REGION Network 6
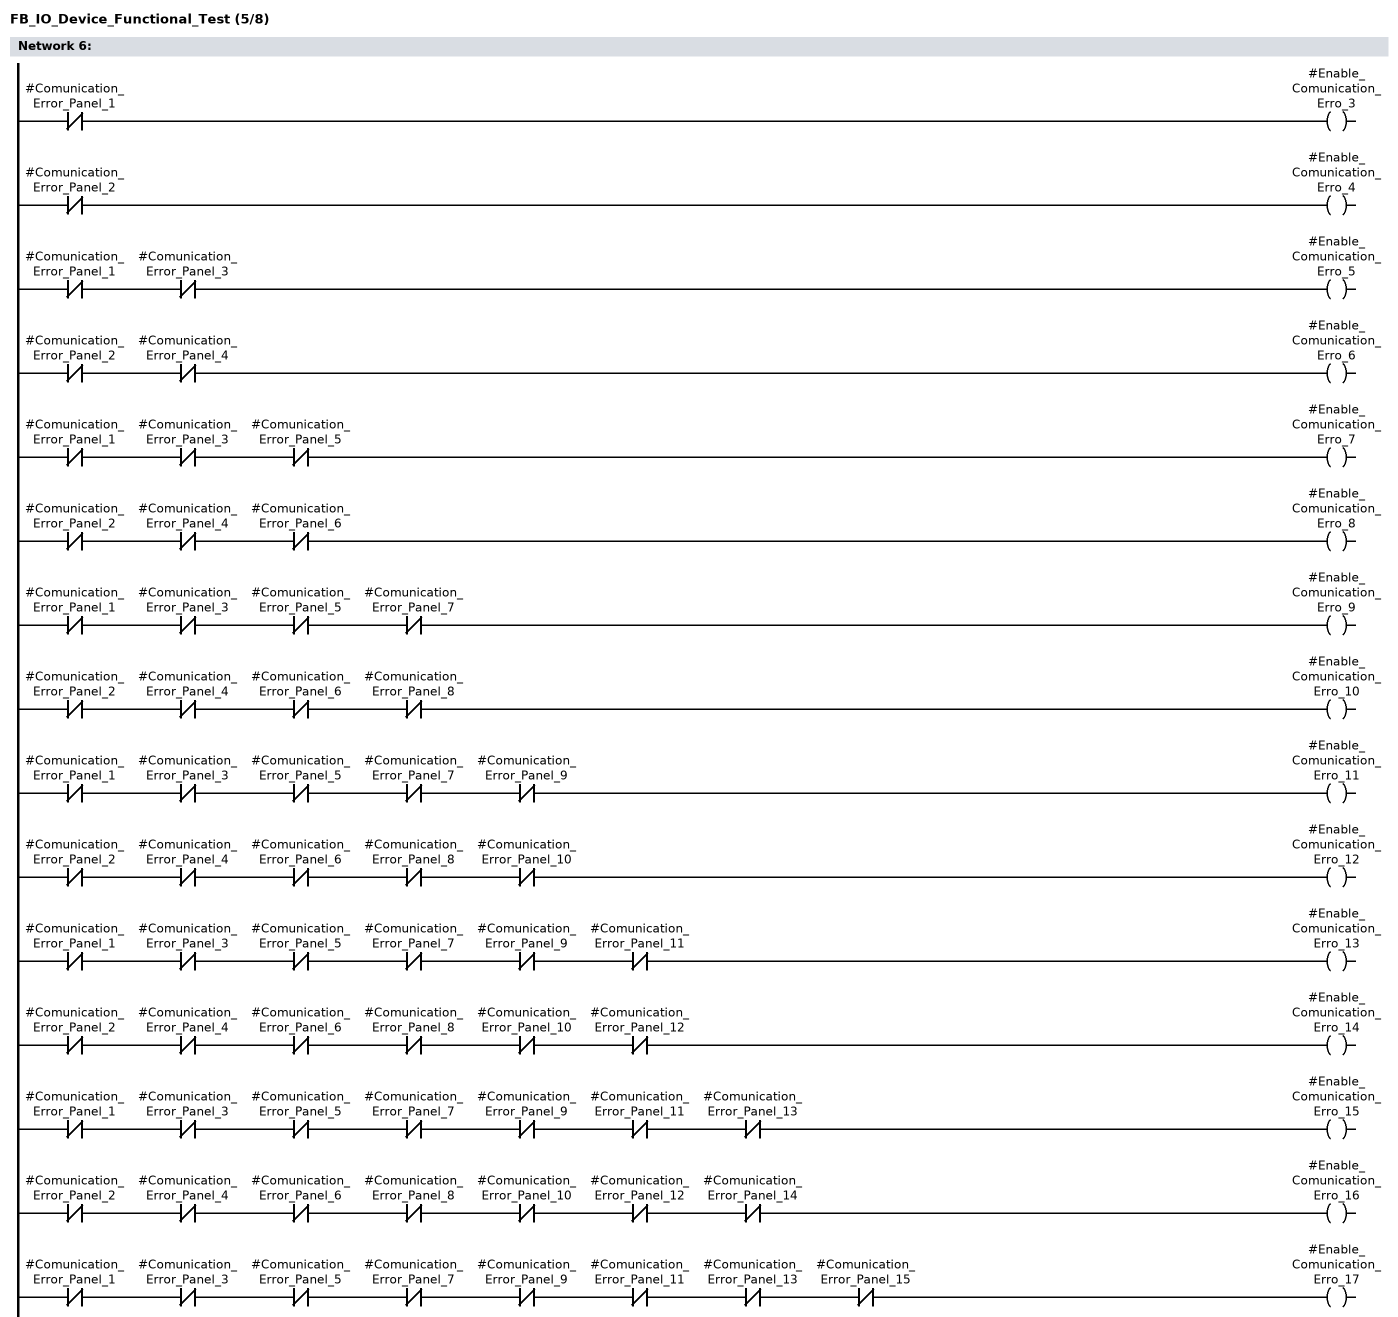
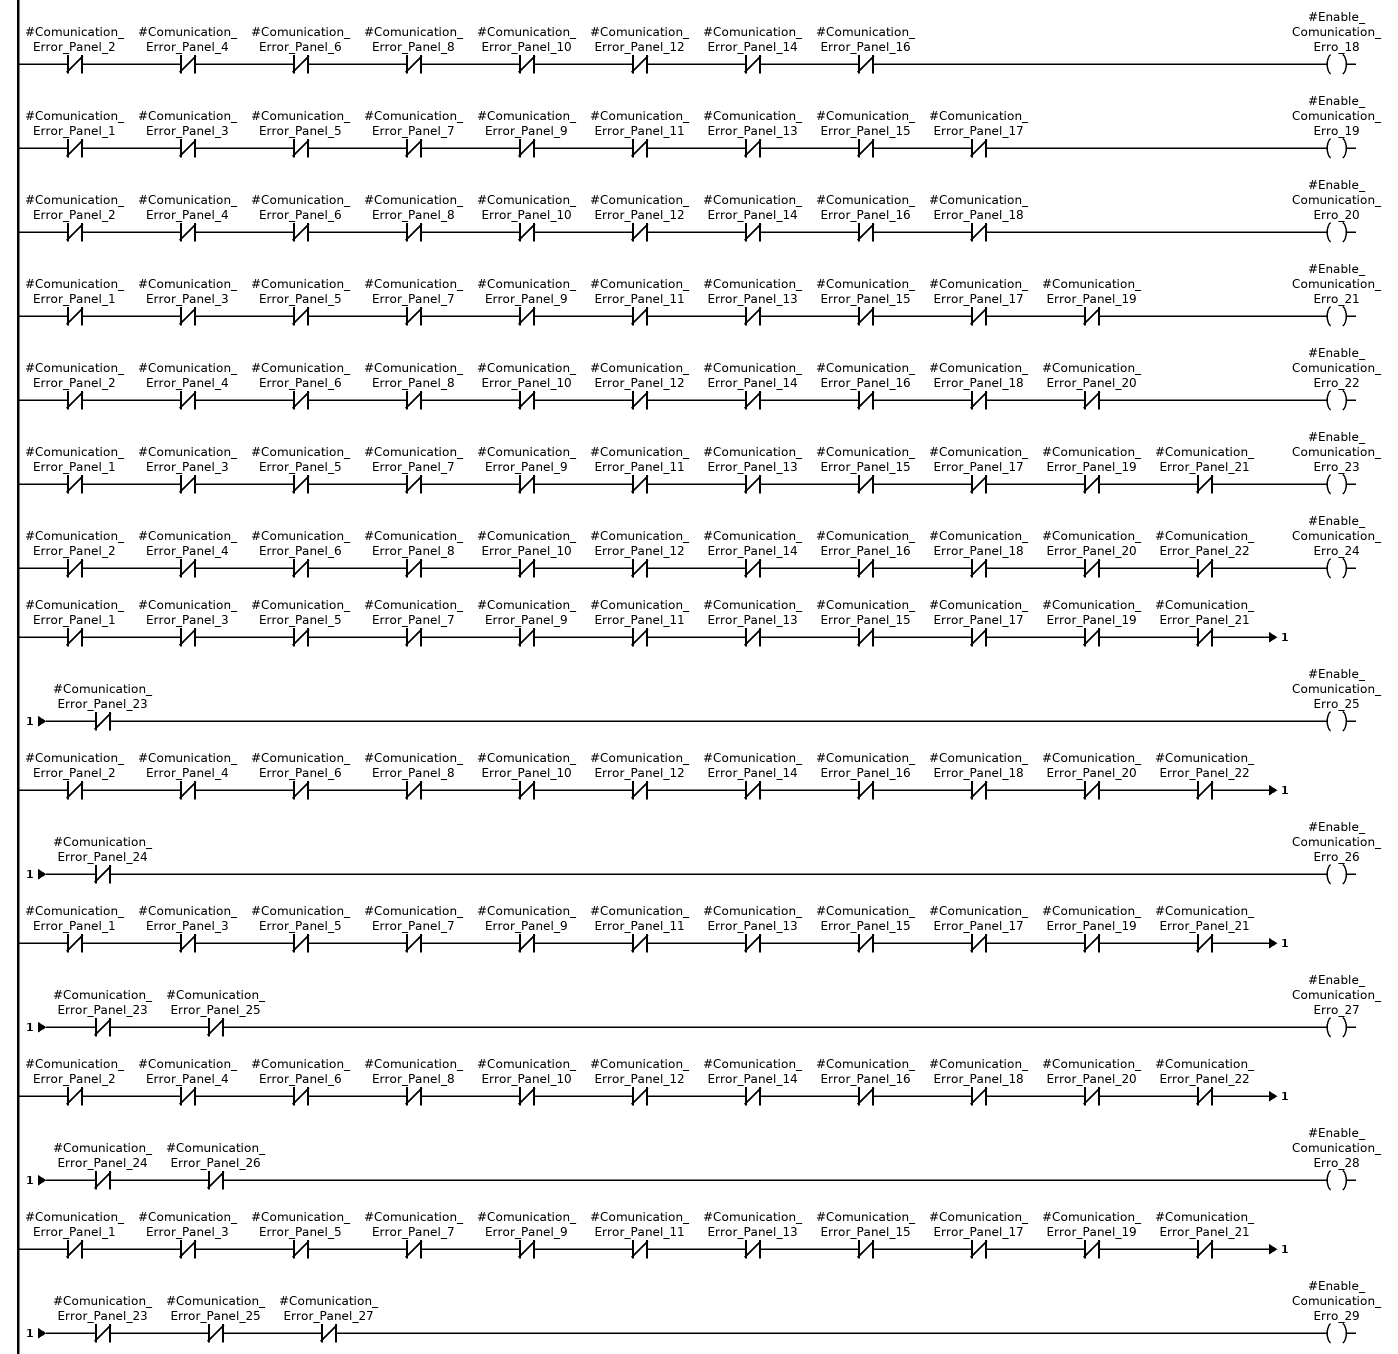
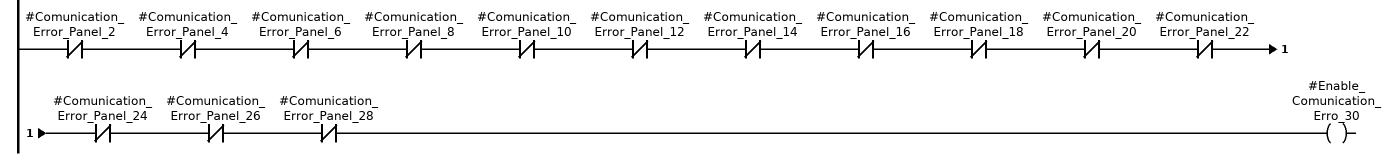
   RUNG wire#powerrail
      I_Contact( #Comunication_Error_Panel_1 )
      Coil( #Enable_Comunication_Erro_3 )
   END_RUNG
   RUNG wire#powerrail
      I_Contact( #Comunication_Error_Panel_2 )
      Coil( #Enable_Comunication_Erro_4 )
   END_RUNG
   RUNG wire#powerrail
      I_Contact( #Comunication_Error_Panel_1 )
      I_Contact( #Comunication_Error_Panel_3 )
      Coil( #Enable_Comunication_Erro_5 )
   END_RUNG
   RUNG wire#powerrail
      I_Contact( #Comunication_Error_Panel_2 )
      I_Contact( #Comunication_Error_Panel_4 )
      Coil( #Enable_Comunication_Erro_6 )
   END_RUNG
   RUNG wire#powerrail
      I_Contact( #Comunication_Error_Panel_1 )
      I_Contact( #Comunication_Error_Panel_3 )
      I_Contact( #Comunication_Error_Panel_5 )
      Coil( #Enable_Comunication_Erro_7 )
   END_RUNG
   RUNG wire#powerrail
      I_Contact( #Comunication_Error_Panel_2 )
      I_Contact( #Comunication_Error_Panel_4 )
      I_Contact( #Comunication_Error_Panel_6 )
      Coil( #Enable_Comunication_Erro_8 )
   END_RUNG
   RUNG wire#powerrail
      I_Contact( #Comunication_Error_Panel_1 )
      I_Contact( #Comunication_Error_Panel_3 )
      I_Contact( #Comunication_Error_Panel_5 )
      I_Contact( #Comunication_Error_Panel_7 )
      Coil( #Enable_Comunication_Erro_9 )
   END_RUNG
   RUNG wire#powerrail
      I_Contact( #Comunication_Error_Panel_2 )
      I_Contact( #Comunication_Error_Panel_4 )
      I_Contact( #Comunication_Error_Panel_6 )
      I_Contact( #Comunication_Error_Panel_8 )
      Coil( #Enable_Comunication_Erro_10 )
   END_RUNG
   RUNG wire#powerrail
      I_Contact( #Comunication_Error_Panel_1 )
      I_Contact( #Comunication_Error_Panel_3 )
      I_Contact( #Comunication_Error_Panel_5 )
      I_Contact( #Comunication_Error_Panel_7 )
      I_Contact( #Comunication_Error_Panel_9 )
      Coil( #Enable_Comunication_Erro_11 )
   END_RUNG
   RUNG wire#powerrail
      I_Contact( #Comunication_Error_Panel_2 )
      I_Contact( #Comunication_Error_Panel_4 )
      I_Contact( #Comunication_Error_Panel_6 )
      I_Contact( #Comunication_Error_Panel_8 )
      I_Contact( #Comunication_Error_Panel_10 )
      Coil( #Enable_Comunication_Erro_12 )
   END_RUNG
   RUNG wire#powerrail
      I_Contact( #Comunication_Error_Panel_1 )
      I_Contact( #Comunication_Error_Panel_3 )
      I_Contact( #Comunication_Error_Panel_5 )
      I_Contact( #Comunication_Error_Panel_7 )
      I_Contact( #Comunication_Error_Panel_9 )
      I_Contact( #Comunication_Error_Panel_11 )
      Coil( #Enable_Comunication_Erro_13 )
   END_RUNG
   RUNG wire#powerrail
      I_Contact( #Comunication_Error_Panel_2 )
      I_Contact( #Comunication_Error_Panel_4 )
      I_Contact( #Comunication_Error_Panel_6 )
      I_Contact( #Comunication_Error_Panel_8 )
      I_Contact( #Comunication_Error_Panel_10 )
      I_Contact( #Comunication_Error_Panel_12 )
      Coil( #Enable_Comunication_Erro_14 )
   END_RUNG
   RUNG wire#powerrail
      I_Contact( #Comunication_Error_Panel_1 )
      I_Contact( #Comunication_Error_Panel_3 )
      I_Contact( #Comunication_Error_Panel_5 )
      I_Contact( #Comunication_Error_Panel_7 )
      I_Contact( #Comunication_Error_Panel_9 )
      I_Contact( #Comunication_Error_Panel_11 )
      I_Contact( #Comunication_Error_Panel_13 )
      Coil( #Enable_Comunication_Erro_15 )
   END_RUNG
   RUNG wire#powerrail
      I_Contact( #Comunication_Error_Panel_2 )
      I_Contact( #Comunication_Error_Panel_4 )
      I_Contact( #Comunication_Error_Panel_6 )
      I_Contact( #Comunication_Error_Panel_8 )
      I_Contact( #Comunication_Error_Panel_10 )
      I_Contact( #Comunication_Error_Panel_12 )
      I_Contact( #Comunication_Error_Panel_14 )
      Coil( #Enable_Comunication_Erro_16 )
   END_RUNG
   RUNG wire#powerrail
      I_Contact( #Comunication_Error_Panel_1 )
      I_Contact( #Comunication_Error_Panel_3 )
      I_Contact( #Comunication_Error_Panel_5 )
      I_Contact( #Comunication_Error_Panel_7 )
      I_Contact( #Comunication_Error_Panel_9 )
      I_Contact( #Comunication_Error_Panel_11 )
      I_Contact( #Comunication_Error_Panel_13 )
      I_Contact( #Comunication_Error_Panel_15 )
      Coil( #Enable_Comunication_Erro_17 )
   END_RUNG
   RUNG wire#powerrail
      I_Contact( #Comunication_Error_Panel_2 )
      I_Contact( #Comunication_Error_Panel_4 )
      I_Contact( #Comunication_Error_Panel_6 )
      I_Contact( #Comunication_Error_Panel_8 )
      I_Contact( #Comunication_Error_Panel_10 )
      I_Contact( #Comunication_Error_Panel_12 )
      I_Contact( #Comunication_Error_Panel_14 )
      I_Contact( #Comunication_Error_Panel_16 )
      Coil( #Enable_Comunication_Erro_18 )
   END_RUNG
   RUNG wire#powerrail
      I_Contact( #Comunication_Error_Panel_1 )
      I_Contact( #Comunication_Error_Panel_3 )
      I_Contact( #Comunication_Error_Panel_5 )
      I_Contact( #Comunication_Error_Panel_7 )
      I_Contact( #Comunication_Error_Panel_9 )
      I_Contact( #Comunication_Error_Panel_11 )
      I_Contact( #Comunication_Error_Panel_13 )
      I_Contact( #Comunication_Error_Panel_15 )
      I_Contact( #Comunication_Error_Panel_17 )
      Coil( #Enable_Comunication_Erro_19 )
   END_RUNG
   RUNG wire#powerrail
      I_Contact( #Comunication_Error_Panel_2 )
      I_Contact( #Comunication_Error_Panel_4 )
      I_Contact( #Comunication_Error_Panel_6 )
      I_Contact( #Comunication_Error_Panel_8 )
      I_Contact( #Comunication_Error_Panel_10 )
      I_Contact( #Comunication_Error_Panel_12 )
      I_Contact( #Comunication_Error_Panel_14 )
      I_Contact( #Comunication_Error_Panel_16 )
      I_Contact( #Comunication_Error_Panel_18 )
      Coil( #Enable_Comunication_Erro_20 )
   END_RUNG
   RUNG wire#powerrail
      I_Contact( #Comunication_Error_Panel_1 )
      I_Contact( #Comunication_Error_Panel_3 )
      I_Contact( #Comunication_Error_Panel_5 )
      I_Contact( #Comunication_Error_Panel_7 )
      I_Contact( #Comunication_Error_Panel_9 )
      I_Contact( #Comunication_Error_Panel_11 )
      I_Contact( #Comunication_Error_Panel_13 )
      I_Contact( #Comunication_Error_Panel_15 )
      I_Contact( #Comunication_Error_Panel_17 )
      I_Contact( #Comunication_Error_Panel_19 )
      Coil( #Enable_Comunication_Erro_21 )
   END_RUNG
   RUNG wire#powerrail
      I_Contact( #Comunication_Error_Panel_2 )
      I_Contact( #Comunication_Error_Panel_4 )
      I_Contact( #Comunication_Error_Panel_6 )
      I_Contact( #Comunication_Error_Panel_8 )
      I_Contact( #Comunication_Error_Panel_10 )
      I_Contact( #Comunication_Error_Panel_12 )
      I_Contact( #Comunication_Error_Panel_14 )
      I_Contact( #Comunication_Error_Panel_16 )
      I_Contact( #Comunication_Error_Panel_18 )
      I_Contact( #Comunication_Error_Panel_20 )
      Coil( #Enable_Comunication_Erro_22 )
   END_RUNG
   RUNG wire#powerrail
      I_Contact( #Comunication_Error_Panel_1 )
      I_Contact( #Comunication_Error_Panel_3 )
      I_Contact( #Comunication_Error_Panel_5 )
      I_Contact( #Comunication_Error_Panel_7 )
      I_Contact( #Comunication_Error_Panel_9 )
      I_Contact( #Comunication_Error_Panel_11 )
      I_Contact( #Comunication_Error_Panel_13 )
      I_Contact( #Comunication_Error_Panel_15 )
      I_Contact( #Comunication_Error_Panel_17 )
      I_Contact( #Comunication_Error_Panel_19 )
      I_Contact( #Comunication_Error_Panel_21 )
      Coil( #Enable_Comunication_Erro_23 )
   END_RUNG
   RUNG wire#powerrail
      I_Contact( #Comunication_Error_Panel_2 )
      I_Contact( #Comunication_Error_Panel_4 )
      I_Contact( #Comunication_Error_Panel_6 )
      I_Contact( #Comunication_Error_Panel_8 )
      I_Contact( #Comunication_Error_Panel_10 )
      I_Contact( #Comunication_Error_Panel_12 )
      I_Contact( #Comunication_Error_Panel_14 )
      I_Contact( #Comunication_Error_Panel_16 )
      I_Contact( #Comunication_Error_Panel_18 )
      I_Contact( #Comunication_Error_Panel_20 )
      I_Contact( #Comunication_Error_Panel_22 )
      Coil( #Enable_Comunication_Erro_24 )
   END_RUNG
   RUNG wire#powerrail
      I_Contact( #Comunication_Error_Panel_1 )
      I_Contact( #Comunication_Error_Panel_3 )
      I_Contact( #Comunication_Error_Panel_5 )
      I_Contact( #Comunication_Error_Panel_7 )
      I_Contact( #Comunication_Error_Panel_9 )
      I_Contact( #Comunication_Error_Panel_11 )
      I_Contact( #Comunication_Error_Panel_13 )
      I_Contact( #Comunication_Error_Panel_15 )
      I_Contact( #Comunication_Error_Panel_17 )
      I_Contact( #Comunication_Error_Panel_19 )
      I_Contact( #Comunication_Error_Panel_21 )
      I_Contact( #Comunication_Error_Panel_23 )
      Coil( #Enable_Comunication_Erro_25 )
   END_RUNG
   RUNG wire#powerrail
      I_Contact( #Comunication_Error_Panel_2 )
      I_Contact( #Comunication_Error_Panel_4 )
      I_Contact( #Comunication_Error_Panel_6 )
      I_Contact( #Comunication_Error_Panel_8 )
      I_Contact( #Comunication_Error_Panel_10 )
      I_Contact( #Comunication_Error_Panel_12 )
      I_Contact( #Comunication_Error_Panel_14 )
      I_Contact( #Comunication_Error_Panel_16 )
      I_Contact( #Comunication_Error_Panel_18 )
      I_Contact( #Comunication_Error_Panel_20 )
      I_Contact( #Comunication_Error_Panel_22 )
      I_Contact( #Comunication_Error_Panel_24 )
      Coil( #Enable_Comunication_Erro_26 )
   END_RUNG
   RUNG wire#powerrail
      I_Contact( #Comunication_Error_Panel_1 )
      I_Contact( #Comunication_Error_Panel_3 )
      I_Contact( #Comunication_Error_Panel_5 )
      I_Contact( #Comunication_Error_Panel_7 )
      I_Contact( #Comunication_Error_Panel_9 )
      I_Contact( #Comunication_Error_Panel_11 )
      I_Contact( #Comunication_Error_Panel_13 )
      I_Contact( #Comunication_Error_Panel_15 )
      I_Contact( #Comunication_Error_Panel_17 )
      I_Contact( #Comunication_Error_Panel_19 )
      I_Contact( #Comunication_Error_Panel_21 )
      I_Contact( #Comunication_Error_Panel_23 )
      I_Contact( #Comunication_Error_Panel_25 )
      Coil( #Enable_Comunication_Erro_27 )
   END_RUNG
   RUNG wire#powerrail
      I_Contact( #Comunication_Error_Panel_2 )
      I_Contact( #Comunication_Error_Panel_4 )
      I_Contact( #Comunication_Error_Panel_6 )
      I_Contact( #Comunication_Error_Panel_8 )
      I_Contact( #Comunication_Error_Panel_10 )
      I_Contact( #Comunication_Error_Panel_12 )
      I_Contact( #Comunication_Error_Panel_14 )
      I_Contact( #Comunication_Error_Panel_16 )
      I_Contact( #Comunication_Error_Panel_18 )
      I_Contact( #Comunication_Error_Panel_20 )
      I_Contact( #Comunication_Error_Panel_22 )
      I_Contact( #Comunication_Error_Panel_24 )
      I_Contact( #Comunication_Error_Panel_26 )
      Coil( #Enable_Comunication_Erro_28 )
   END_RUNG
   RUNG wire#powerrail
      I_Contact( #Comunication_Error_Panel_1 )
      I_Contact( #Comunication_Error_Panel_3 )
      I_Contact( #Comunication_Error_Panel_5 )
      I_Contact( #Comunication_Error_Panel_7 )
      I_Contact( #Comunication_Error_Panel_9 )
      I_Contact( #Comunication_Error_Panel_11 )
      I_Contact( #Comunication_Error_Panel_13 )
      I_Contact( #Comunication_Error_Panel_15 )
      I_Contact( #Comunication_Error_Panel_17 )
      I_Contact( #Comunication_Error_Panel_19 )
      I_Contact( #Comunication_Error_Panel_21 )
      I_Contact( #Comunication_Error_Panel_23 )
      I_Contact( #Comunication_Error_Panel_25 )
      I_Contact( #Comunication_Error_Panel_27 )
      Coil( #Enable_Comunication_Erro_29 )
   END_RUNG
   RUNG wire#powerrail
      I_Contact( #Comunication_Error_Panel_2 )
      I_Contact( #Comunication_Error_Panel_4 )
      I_Contact( #Comunication_Error_Panel_6 )
      I_Contact( #Comunication_Error_Panel_8 )
      I_Contact( #Comunication_Error_Panel_10 )
      I_Contact( #Comunication_Error_Panel_12 )
      I_Contact( #Comunication_Error_Panel_14 )
      I_Contact( #Comunication_Error_Panel_16 )
      I_Contact( #Comunication_Error_Panel_18 )
      I_Contact( #Comunication_Error_Panel_20 )
      I_Contact( #Comunication_Error_Panel_22 )
      I_Contact( #Comunication_Error_Panel_24 )
      I_Contact( #Comunication_Error_Panel_26 )
      I_Contact( #Comunication_Error_Panel_28 )
      Coil( #Enable_Comunication_Erro_30 )
   END_RUNG
   // the same network as SCL:
   #Enable_Comunication_Erro_3 := NOT #Comunication_Error_Panel_1;
   #Enable_Comunication_Erro_4 := NOT #Comunication_Error_Panel_2;
   #Enable_Comunication_Erro_5 := NOT #Comunication_Error_Panel_1 AND NOT #Comunication_Error_Panel_3;
   #Enable_Comunication_Erro_6 := NOT #Comunication_Error_Panel_2 AND NOT #Comunication_Error_Panel_4;
   #Enable_Comunication_Erro_7 := NOT #Comunication_Error_Panel_1 AND NOT #Comunication_Error_Panel_3 AND NOT #Comunication_Error_Panel_5;
   #Enable_Comunication_Erro_8 := NOT #Comunication_Error_Panel_2 AND NOT #Comunication_Error_Panel_4 AND NOT #Comunication_Error_Panel_6;
   #Enable_Comunication_Erro_9 := NOT #Comunication_Error_Panel_1 AND NOT #Comunication_Error_Panel_3 AND NOT #Comunication_Error_Panel_5 AND NOT #Comunication_Error_Panel_7;
   #Enable_Comunication_Erro_10 := NOT #Comunication_Error_Panel_2 AND NOT #Comunication_Error_Panel_4 AND NOT #Comunication_Error_Panel_6 AND NOT #Comunication_Error_Panel_8;
   #Enable_Comunication_Erro_11 := NOT #Comunication_Error_Panel_1 AND NOT #Comunication_Error_Panel_3 AND NOT #Comunication_Error_Panel_5 AND NOT #Comunication_Error_Panel_7 AND NOT #Comunication_Error_Panel_9;
   #Enable_Comunication_Erro_12 := NOT #Comunication_Error_Panel_2 AND NOT #Comunication_Error_Panel_4 AND NOT #Comunication_Error_Panel_6 AND NOT #Comunication_Error_Panel_8 AND NOT #Comunication_Error_Panel_10;
   #Enable_Comunication_Erro_13 := NOT #Comunication_Error_Panel_1 AND NOT #Comunication_Error_Panel_3 AND NOT #Comunication_Error_Panel_5 AND NOT #Comunication_Error_Panel_7 AND NOT #Comunication_Error_Panel_9 AND NOT #Comunication_Error_Panel_11;
   #Enable_Comunication_Erro_14 := NOT #Comunication_Error_Panel_2 AND NOT #Comunication_Error_Panel_4 AND NOT #Comunication_Error_Panel_6 AND NOT #Comunication_Error_Panel_8 AND NOT #Comunication_Error_Panel_10 AND NOT #Comunication_Error_Panel_12;
   #Enable_Comunication_Erro_15 := NOT #Comunication_Error_Panel_1 AND NOT #Comunication_Error_Panel_3 AND NOT #Comunication_Error_Panel_5 AND NOT #Comunication_Error_Panel_7 AND NOT #Comunication_Error_Panel_9 AND NOT #Comunication_Error_Panel_11 AND NOT #Comunication_Error_Panel_13;
   #Enable_Comunication_Erro_16 := NOT #Comunication_Error_Panel_2 AND NOT #Comunication_Error_Panel_4 AND NOT #Comunication_Error_Panel_6 AND NOT #Comunication_Error_Panel_8 AND NOT #Comunication_Error_Panel_10 AND NOT #Comunication_Error_Panel_12 AND NOT #Comunication_Error_Panel_14;
   #Enable_Comunication_Erro_17 := NOT #Comunication_Error_Panel_1 AND NOT #Comunication_Error_Panel_3 AND NOT #Comunication_Error_Panel_5 AND NOT #Comunication_Error_Panel_7 AND NOT #Comunication_Error_Panel_9 AND NOT #Comunication_Error_Panel_11 AND NOT #Comunication_Error_Panel_13 AND NOT #Comunication_Error_Panel_15;
   #Enable_Comunication_Erro_18 := NOT #Comunication_Error_Panel_2 AND NOT #Comunication_Error_Panel_4 AND NOT #Comunication_Error_Panel_6 AND NOT #Comunication_Error_Panel_8 AND NOT #Comunication_Error_Panel_10 AND NOT #Comunication_Error_Panel_12 AND NOT #Comunication_Error_Panel_14 AND NOT #Comunication_Error_Panel_16;
   #Enable_Comunication_Erro_19 := NOT #Comunication_Error_Panel_1 AND NOT #Comunication_Error_Panel_3 AND NOT #Comunication_Error_Panel_5 AND NOT #Comunication_Error_Panel_7 AND NOT #Comunication_Error_Panel_9 AND NOT #Comunication_Error_Panel_11 AND NOT #Comunication_Error_Panel_13 AND NOT #Comunication_Error_Panel_15 AND NOT #Comunication_Error_Panel_17;
   #Enable_Comunication_Erro_20 := NOT #Comunication_Error_Panel_2 AND NOT #Comunication_Error_Panel_4 AND NOT #Comunication_Error_Panel_6 AND NOT #Comunication_Error_Panel_8 AND NOT #Comunication_Error_Panel_10 AND NOT #Comunication_Error_Panel_12 AND NOT #Comunication_Error_Panel_14 AND NOT #Comunication_Error_Panel_16 AND NOT #Comunication_Error_Panel_18;
   #Enable_Comunication_Erro_21 := NOT #Comunication_Error_Panel_1 AND NOT #Comunication_Error_Panel_3 AND NOT #Comunication_Error_Panel_5 AND NOT #Comunication_Error_Panel_7 AND NOT #Comunication_Error_Panel_9 AND NOT #Comunication_Error_Panel_11 AND NOT #Comunication_Error_Panel_13 AND NOT #Comunication_Error_Panel_15 AND NOT #Comunication_Error_Panel_17 AND NOT #Comunication_Error_Panel_19;
   #Enable_Comunication_Erro_22 := NOT #Comunication_Error_Panel_2 AND NOT #Comunication_Error_Panel_4 AND NOT #Comunication_Error_Panel_6 AND NOT #Comunication_Error_Panel_8 AND NOT #Comunication_Error_Panel_10 AND NOT #Comunication_Error_Panel_12 AND NOT #Comunication_Error_Panel_14 AND NOT #Comunication_Error_Panel_16 AND NOT #Comunication_Error_Panel_18 AND NOT #Comunication_Error_Panel_20;
   #Enable_Comunication_Erro_23 := NOT #Comunication_Error_Panel_1 AND NOT #Comunication_Error_Panel_3 AND NOT #Comunication_Error_Panel_5 AND NOT #Comunication_Error_Panel_7 AND NOT #Comunication_Error_Panel_9 AND NOT #Comunication_Error_Panel_11 AND NOT #Comunication_Error_Panel_13 AND NOT #Comunication_Error_Panel_15 AND NOT #Comunication_Error_Panel_17 AND NOT #Comunication_Error_Panel_19 AND NOT #Comunication_Error_Panel_21;
   #Enable_Comunication_Erro_24 := NOT #Comunication_Error_Panel_2 AND NOT #Comunication_Error_Panel_4 AND NOT #Comunication_Error_Panel_6 AND NOT #Comunication_Error_Panel_8 AND NOT #Comunication_Error_Panel_10 AND NOT #Comunication_Error_Panel_12 AND NOT #Comunication_Error_Panel_14 AND NOT #Comunication_Error_Panel_16 AND NOT #Comunication_Error_Panel_18 AND NOT #Comunication_Error_Panel_20 AND NOT #Comunication_Error_Panel_22;
   #Enable_Comunication_Erro_25 := NOT #Comunication_Error_Panel_1 AND NOT #Comunication_Error_Panel_3 AND NOT #Comunication_Error_Panel_5 AND NOT #Comunication_Error_Panel_7 AND NOT #Comunication_Error_Panel_9 AND NOT #Comunication_Error_Panel_11 AND NOT #Comunication_Error_Panel_13 AND NOT #Comunication_Error_Panel_15 AND NOT #Comunication_Error_Panel_17 AND NOT #Comunication_Error_Panel_19 AND NOT #Comunication_Error_Panel_21 AND NOT #Comunication_Error_Panel_23;
   #Enable_Comunication_Erro_26 := NOT #Comunication_Error_Panel_2 AND NOT #Comunication_Error_Panel_4 AND NOT #Comunication_Error_Panel_6 AND NOT #Comunication_Error_Panel_8 AND NOT #Comunication_Error_Panel_10 AND NOT #Comunication_Error_Panel_12 AND NOT #Comunication_Error_Panel_14 AND NOT #Comunication_Error_Panel_16 AND NOT #Comunication_Error_Panel_18 AND NOT #Comunication_Error_Panel_20 AND NOT #Comunication_Error_Panel_22 AND NOT #Comunication_Error_Panel_24;
   #Enable_Comunication_Erro_27 := NOT #Comunication_Error_Panel_1 AND NOT #Comunication_Error_Panel_3 AND NOT #Comunication_Error_Panel_5 AND NOT #Comunication_Error_Panel_7 AND NOT #Comunication_Error_Panel_9 AND NOT #Comunication_Error_Panel_11 AND NOT #Comunication_Error_Panel_13 AND NOT #Comunication_Error_Panel_15 AND NOT #Comunication_Error_Panel_17 AND NOT #Comunication_Error_Panel_19 AND NOT #Comunication_Error_Panel_21 AND NOT #Comunication_Error_Panel_23 AND NOT #Comunication_Error_Panel_25;
   #Enable_Comunication_Erro_28 := NOT #Comunication_Error_Panel_2 AND NOT #Comunication_Error_Panel_4 AND NOT #Comunication_Error_Panel_6 AND NOT #Comunication_Error_Panel_8 AND NOT #Comunication_Error_Panel_10 AND NOT #Comunication_Error_Panel_12 AND NOT #Comunication_Error_Panel_14 AND NOT #Comunication_Error_Panel_16 AND NOT #Comunication_Error_Panel_18 AND NOT #Comunication_Error_Panel_20 AND NOT #Comunication_Error_Panel_22 AND NOT #Comunication_Error_Panel_24 AND NOT #Comunication_Error_Panel_26;
   #Enable_Comunication_Erro_29 := NOT #Comunication_Error_Panel_1 AND NOT #Comunication_Error_Panel_3 AND NOT #Comunication_Error_Panel_5 AND NOT #Comunication_Error_Panel_7 AND NOT #Comunication_Error_Panel_9 AND NOT #Comunication_Error_Panel_11 AND NOT #Comunication_Error_Panel_13 AND NOT #Comunication_Error_Panel_15 AND NOT #Comunication_Error_Panel_17 AND NOT #Comunication_Error_Panel_19 AND NOT #Comunication_Error_Panel_21 AND NOT #Comunication_Error_Panel_23 AND NOT #Comunication_Error_Panel_25 AND NOT #Comunication_Error_Panel_27;
   #Enable_Comunication_Erro_30 := NOT #Comunication_Error_Panel_2 AND NOT #Comunication_Error_Panel_4 AND NOT #Comunication_Error_Panel_6 AND NOT #Comunication_Error_Panel_8 AND NOT #Comunication_Error_Panel_10 AND NOT #Comunication_Error_Panel_12 AND NOT #Comunication_Error_Panel_14 AND NOT #Comunication_Error_Panel_16 AND NOT #Comunication_Error_Panel_18 AND NOT #Comunication_Error_Panel_20 AND NOT #Comunication_Error_Panel_22 AND NOT #Comunication_Error_Panel_24 AND NOT #Comunication_Error_Panel_26 AND NOT #Comunication_Error_Panel_28;
END_REGION

REGION Network 7
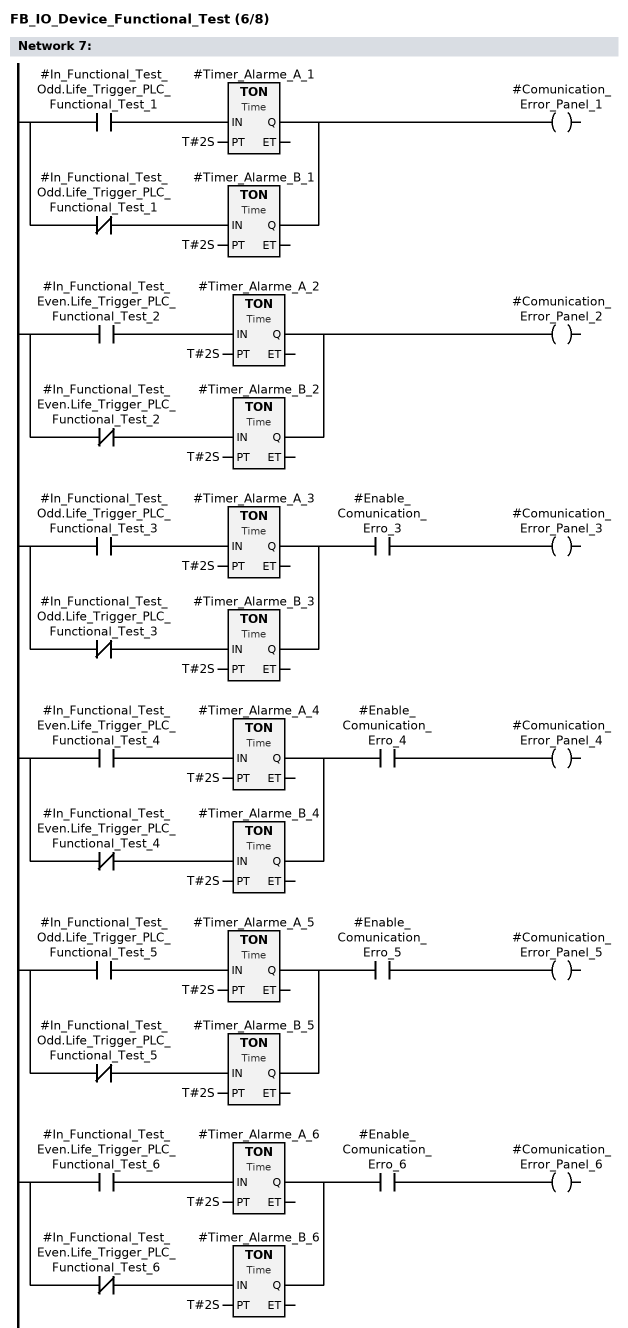
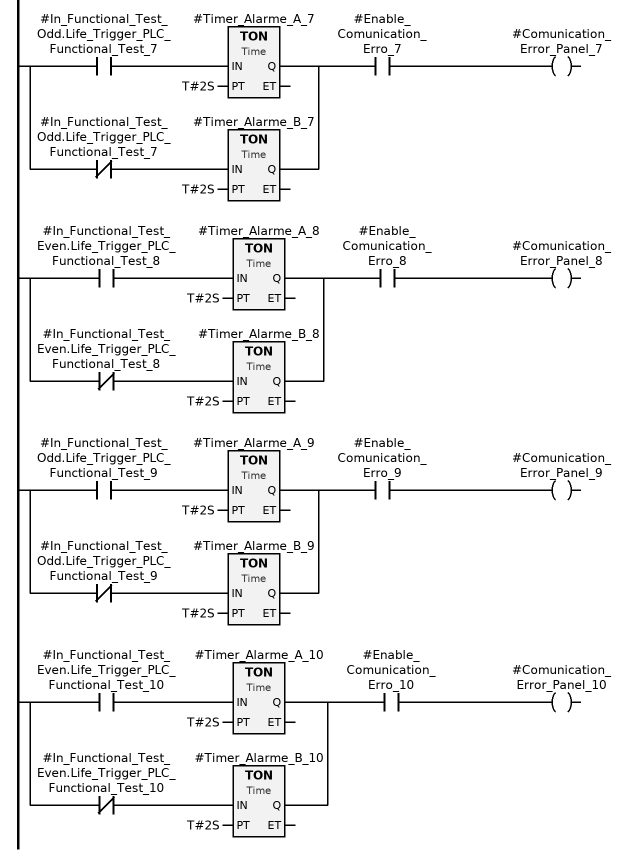
   RUNG wire#powerrail
      Contact( #In_Functional_Test_Odd.Life_Trigger_PLC_Functional_Test_1 )
      { S7_Templates := "time_type := Time" } #Timer_Alarme_A_1.TON(pt := T#2S, et =>)
      wire#w1
      Coil( #Comunication_Error_Panel_1 )
   END_RUNG
   RUNG wire#powerrail
      I_Contact( #In_Functional_Test_Odd.Life_Trigger_PLC_Functional_Test_1 )
      { S7_Templates := "time_type := Time" } #Timer_Alarme_B_1.TON(pt := T#2S, et =>)
   END_RUNG wire#w1
   RUNG wire#powerrail
      Contact( #In_Functional_Test_Even.Life_Trigger_PLC_Functional_Test_2 )
      { S7_Templates := "time_type := Time" } #Timer_Alarme_A_2.TON(pt := T#2S, et =>)
      wire#w2
      Coil( #Comunication_Error_Panel_2 )
   END_RUNG
   RUNG wire#powerrail
      I_Contact( #In_Functional_Test_Even.Life_Trigger_PLC_Functional_Test_2 )
      { S7_Templates := "time_type := Time" } #Timer_Alarme_B_2.TON(pt := T#2S, et =>)
   END_RUNG wire#w2
   RUNG wire#powerrail
      Contact( #In_Functional_Test_Odd.Life_Trigger_PLC_Functional_Test_3 )
      { S7_Templates := "time_type := Time" } #Timer_Alarme_A_3.TON(pt := T#2S, et =>)
      wire#w3
      Contact( #Enable_Comunication_Erro_3 )
      Coil( #Comunication_Error_Panel_3 )
   END_RUNG
   RUNG wire#powerrail
      I_Contact( #In_Functional_Test_Odd.Life_Trigger_PLC_Functional_Test_3 )
      { S7_Templates := "time_type := Time" } #Timer_Alarme_B_3.TON(pt := T#2S, et =>)
   END_RUNG wire#w3
   RUNG wire#powerrail
      Contact( #In_Functional_Test_Even.Life_Trigger_PLC_Functional_Test_4 )
      { S7_Templates := "time_type := Time" } #Timer_Alarme_A_4.TON(pt := T#2S, et =>)
      wire#w4
      Contact( #Enable_Comunication_Erro_4 )
      Coil( #Comunication_Error_Panel_4 )
   END_RUNG
   RUNG wire#powerrail
      I_Contact( #In_Functional_Test_Even.Life_Trigger_PLC_Functional_Test_4 )
      { S7_Templates := "time_type := Time" } #Timer_Alarme_B_4.TON(pt := T#2S, et =>)
   END_RUNG wire#w4
   RUNG wire#powerrail
      Contact( #In_Functional_Test_Odd.Life_Trigger_PLC_Functional_Test_5 )
      { S7_Templates := "time_type := Time" } #Timer_Alarme_A_5.TON(pt := T#2S, et =>)
      wire#w5
      Contact( #Enable_Comunication_Erro_5 )
      Coil( #Comunication_Error_Panel_5 )
   END_RUNG
   RUNG wire#powerrail
      I_Contact( #In_Functional_Test_Odd.Life_Trigger_PLC_Functional_Test_5 )
      { S7_Templates := "time_type := Time" } #Timer_Alarme_B_5.TON(pt := T#2S, et =>)
   END_RUNG wire#w5
   RUNG wire#powerrail
      Contact( #In_Functional_Test_Even.Life_Trigger_PLC_Functional_Test_6 )
      { S7_Templates := "time_type := Time" } #Timer_Alarme_A_6.TON(pt := T#2S, et =>)
      wire#w6
      Contact( #Enable_Comunication_Erro_6 )
      Coil( #Comunication_Error_Panel_6 )
   END_RUNG
   RUNG wire#powerrail
      I_Contact( #In_Functional_Test_Even.Life_Trigger_PLC_Functional_Test_6 )
      { S7_Templates := "time_type := Time" } #Timer_Alarme_B_6.TON(pt := T#2S, et =>)
   END_RUNG wire#w6
   RUNG wire#powerrail
      Contact( #In_Functional_Test_Odd.Life_Trigger_PLC_Functional_Test_7 )
      { S7_Templates := "time_type := Time" } #Timer_Alarme_A_7.TON(pt := T#2S, et =>)
      wire#w7
      Contact( #Enable_Comunication_Erro_7 )
      Coil( #Comunication_Error_Panel_7 )
   END_RUNG
   RUNG wire#powerrail
      I_Contact( #In_Functional_Test_Odd.Life_Trigger_PLC_Functional_Test_7 )
      { S7_Templates := "time_type := Time" } #Timer_Alarme_B_7.TON(pt := T#2S, et =>)
   END_RUNG wire#w7
   RUNG wire#powerrail
      Contact( #In_Functional_Test_Even.Life_Trigger_PLC_Functional_Test_8 )
      { S7_Templates := "time_type := Time" } #Timer_Alarme_A_8.TON(pt := T#2S, et =>)
      wire#w8
      Contact( #Enable_Comunication_Erro_8 )
      Coil( #Comunication_Error_Panel_8 )
   END_RUNG
   RUNG wire#powerrail
      I_Contact( #In_Functional_Test_Even.Life_Trigger_PLC_Functional_Test_8 )
      { S7_Templates := "time_type := Time" } #Timer_Alarme_B_8.TON(pt := T#2S, et =>)
   END_RUNG wire#w8
   RUNG wire#powerrail
      Contact( #In_Functional_Test_Odd.Life_Trigger_PLC_Functional_Test_9 )
      { S7_Templates := "time_type := Time" } #Timer_Alarme_A_9.TON(pt := T#2S, et =>)
      wire#w9
      Contact( #Enable_Comunication_Erro_9 )
      Coil( #Comunication_Error_Panel_9 )
   END_RUNG
   RUNG wire#powerrail
      I_Contact( #In_Functional_Test_Odd.Life_Trigger_PLC_Functional_Test_9 )
      { S7_Templates := "time_type := Time" } #Timer_Alarme_B_9.TON(pt := T#2S, et =>)
   END_RUNG wire#w9
   RUNG wire#powerrail
      Contact( #In_Functional_Test_Even.Life_Trigger_PLC_Functional_Test_10 )
      { S7_Templates := "time_type := Time" } #Timer_Alarme_A_10.TON(pt := T#2S, et =>)
      wire#w10
      Contact( #Enable_Comunication_Erro_10 )
      Coil( #Comunication_Error_Panel_10 )
   END_RUNG
   RUNG wire#powerrail
      I_Contact( #In_Functional_Test_Even.Life_Trigger_PLC_Functional_Test_10 )
      { S7_Templates := "time_type := Time" } #Timer_Alarme_B_10.TON(pt := T#2S, et =>)
   END_RUNG wire#w10
   // the same network as SCL:
   #Timer_Alarme_A_1(IN := #In_Functional_Test_Odd.Life_Trigger_PLC_Functional_Test_1, PT := T#2S);   // TON
   #Timer_Alarme_B_1(IN := NOT #In_Functional_Test_Odd.Life_Trigger_PLC_Functional_Test_1, PT := T#2S);   // TON
   #Comunication_Error_Panel_1 := #Timer_Alarme_A_1.Q OR #Timer_Alarme_B_1.Q;
   #Timer_Alarme_A_2(IN := #In_Functional_Test_Even.Life_Trigger_PLC_Functional_Test_2, PT := T#2S);   // TON
   #Timer_Alarme_B_2(IN := NOT #In_Functional_Test_Even.Life_Trigger_PLC_Functional_Test_2, PT := T#2S);   // TON
   #Comunication_Error_Panel_2 := #Timer_Alarme_A_2.Q OR #Timer_Alarme_B_2.Q;
   #Timer_Alarme_A_3(IN := #In_Functional_Test_Odd.Life_Trigger_PLC_Functional_Test_3, PT := T#2S);   // TON
   #Timer_Alarme_B_3(IN := NOT #In_Functional_Test_Odd.Life_Trigger_PLC_Functional_Test_3, PT := T#2S);   // TON
   #Comunication_Error_Panel_3 := (#Timer_Alarme_A_3.Q OR #Timer_Alarme_B_3.Q) AND #Enable_Comunication_Erro_3;
   #Timer_Alarme_A_4(IN := #In_Functional_Test_Even.Life_Trigger_PLC_Functional_Test_4, PT := T#2S);   // TON
   #Timer_Alarme_B_4(IN := NOT #In_Functional_Test_Even.Life_Trigger_PLC_Functional_Test_4, PT := T#2S);   // TON
   #Comunication_Error_Panel_4 := (#Timer_Alarme_A_4.Q OR #Timer_Alarme_B_4.Q) AND #Enable_Comunication_Erro_4;
   #Timer_Alarme_A_5(IN := #In_Functional_Test_Odd.Life_Trigger_PLC_Functional_Test_5, PT := T#2S);   // TON
   #Timer_Alarme_B_5(IN := NOT #In_Functional_Test_Odd.Life_Trigger_PLC_Functional_Test_5, PT := T#2S);   // TON
   #Comunication_Error_Panel_5 := (#Timer_Alarme_A_5.Q OR #Timer_Alarme_B_5.Q) AND #Enable_Comunication_Erro_5;
   #Timer_Alarme_A_6(IN := #In_Functional_Test_Even.Life_Trigger_PLC_Functional_Test_6, PT := T#2S);   // TON
   #Timer_Alarme_B_6(IN := NOT #In_Functional_Test_Even.Life_Trigger_PLC_Functional_Test_6, PT := T#2S);   // TON
   #Comunication_Error_Panel_6 := (#Timer_Alarme_A_6.Q OR #Timer_Alarme_B_6.Q) AND #Enable_Comunication_Erro_6;
   #Timer_Alarme_A_7(IN := #In_Functional_Test_Odd.Life_Trigger_PLC_Functional_Test_7, PT := T#2S);   // TON
   #Timer_Alarme_B_7(IN := NOT #In_Functional_Test_Odd.Life_Trigger_PLC_Functional_Test_7, PT := T#2S);   // TON
   #Comunication_Error_Panel_7 := (#Timer_Alarme_A_7.Q OR #Timer_Alarme_B_7.Q) AND #Enable_Comunication_Erro_7;
   #Timer_Alarme_A_8(IN := #In_Functional_Test_Even.Life_Trigger_PLC_Functional_Test_8, PT := T#2S);   // TON
   #Timer_Alarme_B_8(IN := NOT #In_Functional_Test_Even.Life_Trigger_PLC_Functional_Test_8, PT := T#2S);   // TON
   #Comunication_Error_Panel_8 := (#Timer_Alarme_A_8.Q OR #Timer_Alarme_B_8.Q) AND #Enable_Comunication_Erro_8;
   #Timer_Alarme_A_9(IN := #In_Functional_Test_Odd.Life_Trigger_PLC_Functional_Test_9, PT := T#2S);   // TON
   #Timer_Alarme_B_9(IN := NOT #In_Functional_Test_Odd.Life_Trigger_PLC_Functional_Test_9, PT := T#2S);   // TON
   #Comunication_Error_Panel_9 := (#Timer_Alarme_A_9.Q OR #Timer_Alarme_B_9.Q) AND #Enable_Comunication_Erro_9;
   #Timer_Alarme_A_10(IN := #In_Functional_Test_Even.Life_Trigger_PLC_Functional_Test_10, PT := T#2S);   // TON
   #Timer_Alarme_B_10(IN := NOT #In_Functional_Test_Even.Life_Trigger_PLC_Functional_Test_10, PT := T#2S);   // TON
   #Comunication_Error_Panel_10 := (#Timer_Alarme_A_10.Q OR #Timer_Alarme_B_10.Q) AND #Enable_Comunication_Erro_10;
END_REGION

REGION Network 8
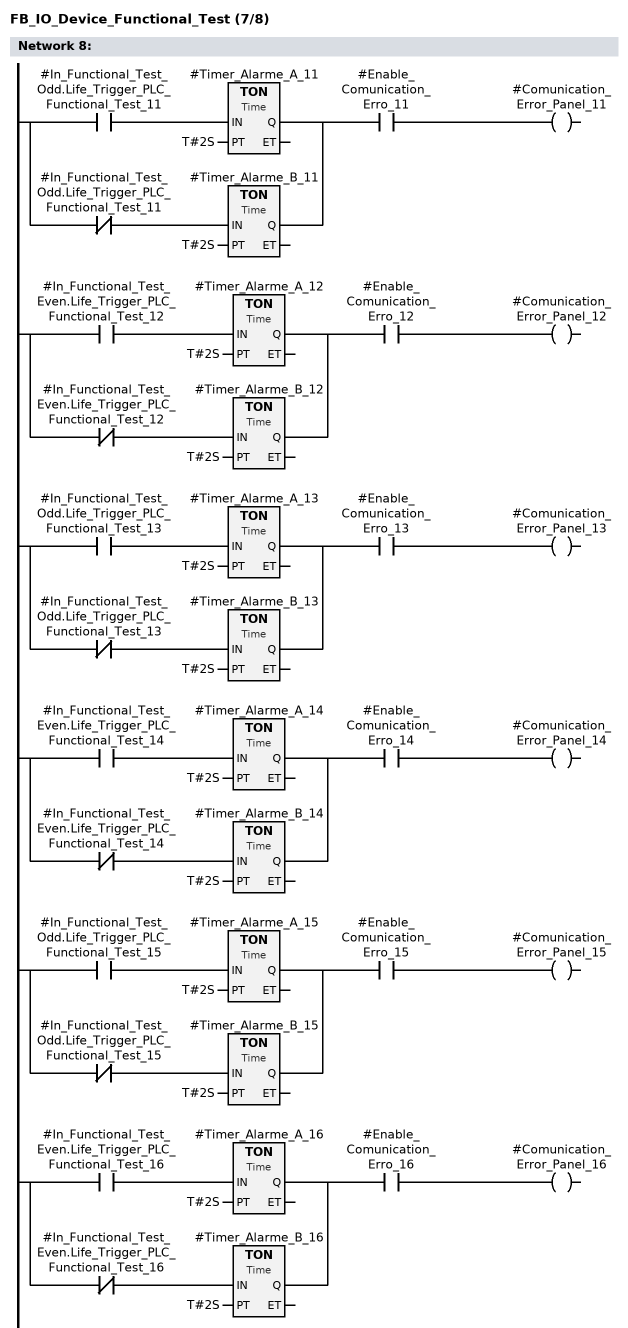
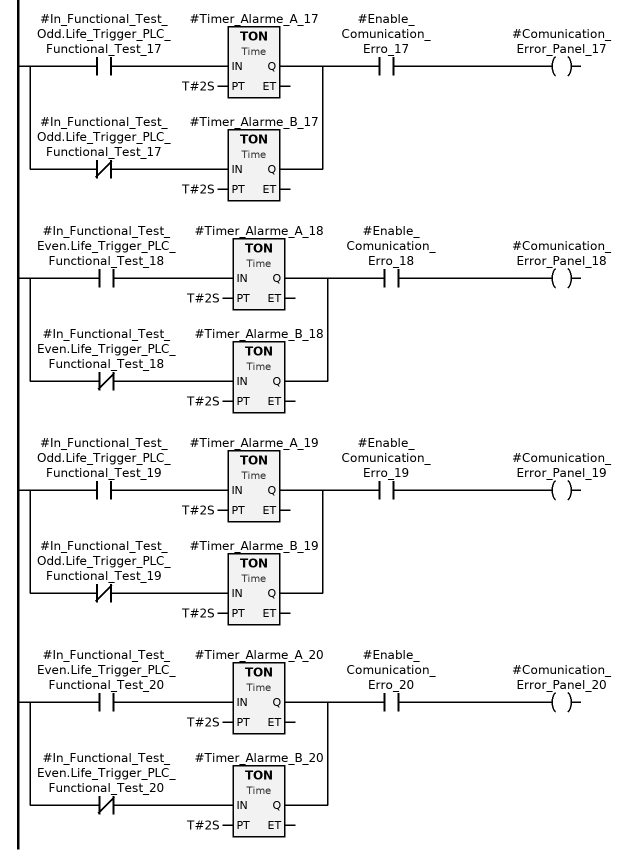
   RUNG wire#powerrail
      Contact( #In_Functional_Test_Odd.Life_Trigger_PLC_Functional_Test_11 )
      { S7_Templates := "time_type := Time" } #Timer_Alarme_A_11.TON(pt := T#2S, et =>)
      wire#w1
      Contact( #Enable_Comunication_Erro_11 )
      Coil( #Comunication_Error_Panel_11 )
   END_RUNG
   RUNG wire#powerrail
      I_Contact( #In_Functional_Test_Odd.Life_Trigger_PLC_Functional_Test_11 )
      { S7_Templates := "time_type := Time" } #Timer_Alarme_B_11.TON(pt := T#2S, et =>)
   END_RUNG wire#w1
   RUNG wire#powerrail
      Contact( #In_Functional_Test_Even.Life_Trigger_PLC_Functional_Test_12 )
      { S7_Templates := "time_type := Time" } #Timer_Alarme_A_12.TON(pt := T#2S, et =>)
      wire#w2
      Contact( #Enable_Comunication_Erro_12 )
      Coil( #Comunication_Error_Panel_12 )
   END_RUNG
   RUNG wire#powerrail
      I_Contact( #In_Functional_Test_Even.Life_Trigger_PLC_Functional_Test_12 )
      { S7_Templates := "time_type := Time" } #Timer_Alarme_B_12.TON(pt := T#2S, et =>)
   END_RUNG wire#w2
   RUNG wire#powerrail
      Contact( #In_Functional_Test_Odd.Life_Trigger_PLC_Functional_Test_13 )
      { S7_Templates := "time_type := Time" } #Timer_Alarme_A_13.TON(pt := T#2S, et =>)
      wire#w3
      Contact( #Enable_Comunication_Erro_13 )
      Coil( #Comunication_Error_Panel_13 )
   END_RUNG
   RUNG wire#powerrail
      I_Contact( #In_Functional_Test_Odd.Life_Trigger_PLC_Functional_Test_13 )
      { S7_Templates := "time_type := Time" } #Timer_Alarme_B_13.TON(pt := T#2S, et =>)
   END_RUNG wire#w3
   RUNG wire#powerrail
      Contact( #In_Functional_Test_Even.Life_Trigger_PLC_Functional_Test_14 )
      { S7_Templates := "time_type := Time" } #Timer_Alarme_A_14.TON(pt := T#2S, et =>)
      wire#w4
      Contact( #Enable_Comunication_Erro_14 )
      Coil( #Comunication_Error_Panel_14 )
   END_RUNG
   RUNG wire#powerrail
      I_Contact( #In_Functional_Test_Even.Life_Trigger_PLC_Functional_Test_14 )
      { S7_Templates := "time_type := Time" } #Timer_Alarme_B_14.TON(pt := T#2S, et =>)
   END_RUNG wire#w4
   RUNG wire#powerrail
      Contact( #In_Functional_Test_Odd.Life_Trigger_PLC_Functional_Test_15 )
      { S7_Templates := "time_type := Time" } #Timer_Alarme_A_15.TON(pt := T#2S, et =>)
      wire#w5
      Contact( #Enable_Comunication_Erro_15 )
      Coil( #Comunication_Error_Panel_15 )
   END_RUNG
   RUNG wire#powerrail
      I_Contact( #In_Functional_Test_Odd.Life_Trigger_PLC_Functional_Test_15 )
      { S7_Templates := "time_type := Time" } #Timer_Alarme_B_15.TON(pt := T#2S, et =>)
   END_RUNG wire#w5
   RUNG wire#powerrail
      Contact( #In_Functional_Test_Even.Life_Trigger_PLC_Functional_Test_16 )
      { S7_Templates := "time_type := Time" } #Timer_Alarme_A_16.TON(pt := T#2S, et =>)
      wire#w6
      Contact( #Enable_Comunication_Erro_16 )
      Coil( #Comunication_Error_Panel_16 )
   END_RUNG
   RUNG wire#powerrail
      I_Contact( #In_Functional_Test_Even.Life_Trigger_PLC_Functional_Test_16 )
      { S7_Templates := "time_type := Time" } #Timer_Alarme_B_16.TON(pt := T#2S, et =>)
   END_RUNG wire#w6
   RUNG wire#powerrail
      Contact( #In_Functional_Test_Odd.Life_Trigger_PLC_Functional_Test_17 )
      { S7_Templates := "time_type := Time" } #Timer_Alarme_A_17.TON(pt := T#2S, et =>)
      wire#w7
      Contact( #Enable_Comunication_Erro_17 )
      Coil( #Comunication_Error_Panel_17 )
   END_RUNG
   RUNG wire#powerrail
      I_Contact( #In_Functional_Test_Odd.Life_Trigger_PLC_Functional_Test_17 )
      { S7_Templates := "time_type := Time" } #Timer_Alarme_B_17.TON(pt := T#2S, et =>)
   END_RUNG wire#w7
   RUNG wire#powerrail
      Contact( #In_Functional_Test_Even.Life_Trigger_PLC_Functional_Test_18 )
      { S7_Templates := "time_type := Time" } #Timer_Alarme_A_18.TON(pt := T#2S, et =>)
      wire#w8
      Contact( #Enable_Comunication_Erro_18 )
      Coil( #Comunication_Error_Panel_18 )
   END_RUNG
   RUNG wire#powerrail
      I_Contact( #In_Functional_Test_Even.Life_Trigger_PLC_Functional_Test_18 )
      { S7_Templates := "time_type := Time" } #Timer_Alarme_B_18.TON(pt := T#2S, et =>)
   END_RUNG wire#w8
   RUNG wire#powerrail
      Contact( #In_Functional_Test_Odd.Life_Trigger_PLC_Functional_Test_19 )
      { S7_Templates := "time_type := Time" } #Timer_Alarme_A_19.TON(pt := T#2S, et =>)
      wire#w9
      Contact( #Enable_Comunication_Erro_19 )
      Coil( #Comunication_Error_Panel_19 )
   END_RUNG
   RUNG wire#powerrail
      I_Contact( #In_Functional_Test_Odd.Life_Trigger_PLC_Functional_Test_19 )
      { S7_Templates := "time_type := Time" } #Timer_Alarme_B_19.TON(pt := T#2S, et =>)
   END_RUNG wire#w9
   RUNG wire#powerrail
      Contact( #In_Functional_Test_Even.Life_Trigger_PLC_Functional_Test_20 )
      { S7_Templates := "time_type := Time" } #Timer_Alarme_A_20.TON(pt := T#2S, et =>)
      wire#w10
      Contact( #Enable_Comunication_Erro_20 )
      Coil( #Comunication_Error_Panel_20 )
   END_RUNG
   RUNG wire#powerrail
      I_Contact( #In_Functional_Test_Even.Life_Trigger_PLC_Functional_Test_20 )
      { S7_Templates := "time_type := Time" } #Timer_Alarme_B_20.TON(pt := T#2S, et =>)
   END_RUNG wire#w10
   // the same network as SCL:
   #Timer_Alarme_A_11(IN := #In_Functional_Test_Odd.Life_Trigger_PLC_Functional_Test_11, PT := T#2S);   // TON
   #Timer_Alarme_B_11(IN := NOT #In_Functional_Test_Odd.Life_Trigger_PLC_Functional_Test_11, PT := T#2S);   // TON
   #Comunication_Error_Panel_11 := (#Timer_Alarme_A_11.Q OR #Timer_Alarme_B_11.Q) AND #Enable_Comunication_Erro_11;
   #Timer_Alarme_A_12(IN := #In_Functional_Test_Even.Life_Trigger_PLC_Functional_Test_12, PT := T#2S);   // TON
   #Timer_Alarme_B_12(IN := NOT #In_Functional_Test_Even.Life_Trigger_PLC_Functional_Test_12, PT := T#2S);   // TON
   #Comunication_Error_Panel_12 := (#Timer_Alarme_A_12.Q OR #Timer_Alarme_B_12.Q) AND #Enable_Comunication_Erro_12;
   #Timer_Alarme_A_13(IN := #In_Functional_Test_Odd.Life_Trigger_PLC_Functional_Test_13, PT := T#2S);   // TON
   #Timer_Alarme_B_13(IN := NOT #In_Functional_Test_Odd.Life_Trigger_PLC_Functional_Test_13, PT := T#2S);   // TON
   #Comunication_Error_Panel_13 := (#Timer_Alarme_A_13.Q OR #Timer_Alarme_B_13.Q) AND #Enable_Comunication_Erro_13;
   #Timer_Alarme_A_14(IN := #In_Functional_Test_Even.Life_Trigger_PLC_Functional_Test_14, PT := T#2S);   // TON
   #Timer_Alarme_B_14(IN := NOT #In_Functional_Test_Even.Life_Trigger_PLC_Functional_Test_14, PT := T#2S);   // TON
   #Comunication_Error_Panel_14 := (#Timer_Alarme_A_14.Q OR #Timer_Alarme_B_14.Q) AND #Enable_Comunication_Erro_14;
   #Timer_Alarme_A_15(IN := #In_Functional_Test_Odd.Life_Trigger_PLC_Functional_Test_15, PT := T#2S);   // TON
   #Timer_Alarme_B_15(IN := NOT #In_Functional_Test_Odd.Life_Trigger_PLC_Functional_Test_15, PT := T#2S);   // TON
   #Comunication_Error_Panel_15 := (#Timer_Alarme_A_15.Q OR #Timer_Alarme_B_15.Q) AND #Enable_Comunication_Erro_15;
   #Timer_Alarme_A_16(IN := #In_Functional_Test_Even.Life_Trigger_PLC_Functional_Test_16, PT := T#2S);   // TON
   #Timer_Alarme_B_16(IN := NOT #In_Functional_Test_Even.Life_Trigger_PLC_Functional_Test_16, PT := T#2S);   // TON
   #Comunication_Error_Panel_16 := (#Timer_Alarme_A_16.Q OR #Timer_Alarme_B_16.Q) AND #Enable_Comunication_Erro_16;
   #Timer_Alarme_A_17(IN := #In_Functional_Test_Odd.Life_Trigger_PLC_Functional_Test_17, PT := T#2S);   // TON
   #Timer_Alarme_B_17(IN := NOT #In_Functional_Test_Odd.Life_Trigger_PLC_Functional_Test_17, PT := T#2S);   // TON
   #Comunication_Error_Panel_17 := (#Timer_Alarme_A_17.Q OR #Timer_Alarme_B_17.Q) AND #Enable_Comunication_Erro_17;
   #Timer_Alarme_A_18(IN := #In_Functional_Test_Even.Life_Trigger_PLC_Functional_Test_18, PT := T#2S);   // TON
   #Timer_Alarme_B_18(IN := NOT #In_Functional_Test_Even.Life_Trigger_PLC_Functional_Test_18, PT := T#2S);   // TON
   #Comunication_Error_Panel_18 := (#Timer_Alarme_A_18.Q OR #Timer_Alarme_B_18.Q) AND #Enable_Comunication_Erro_18;
   #Timer_Alarme_A_19(IN := #In_Functional_Test_Odd.Life_Trigger_PLC_Functional_Test_19, PT := T#2S);   // TON
   #Timer_Alarme_B_19(IN := NOT #In_Functional_Test_Odd.Life_Trigger_PLC_Functional_Test_19, PT := T#2S);   // TON
   #Comunication_Error_Panel_19 := (#Timer_Alarme_A_19.Q OR #Timer_Alarme_B_19.Q) AND #Enable_Comunication_Erro_19;
   #Timer_Alarme_A_20(IN := #In_Functional_Test_Even.Life_Trigger_PLC_Functional_Test_20, PT := T#2S);   // TON
   #Timer_Alarme_B_20(IN := NOT #In_Functional_Test_Even.Life_Trigger_PLC_Functional_Test_20, PT := T#2S);   // TON
   #Comunication_Error_Panel_20 := (#Timer_Alarme_A_20.Q OR #Timer_Alarme_B_20.Q) AND #Enable_Comunication_Erro_20;
END_REGION

REGION Network 9
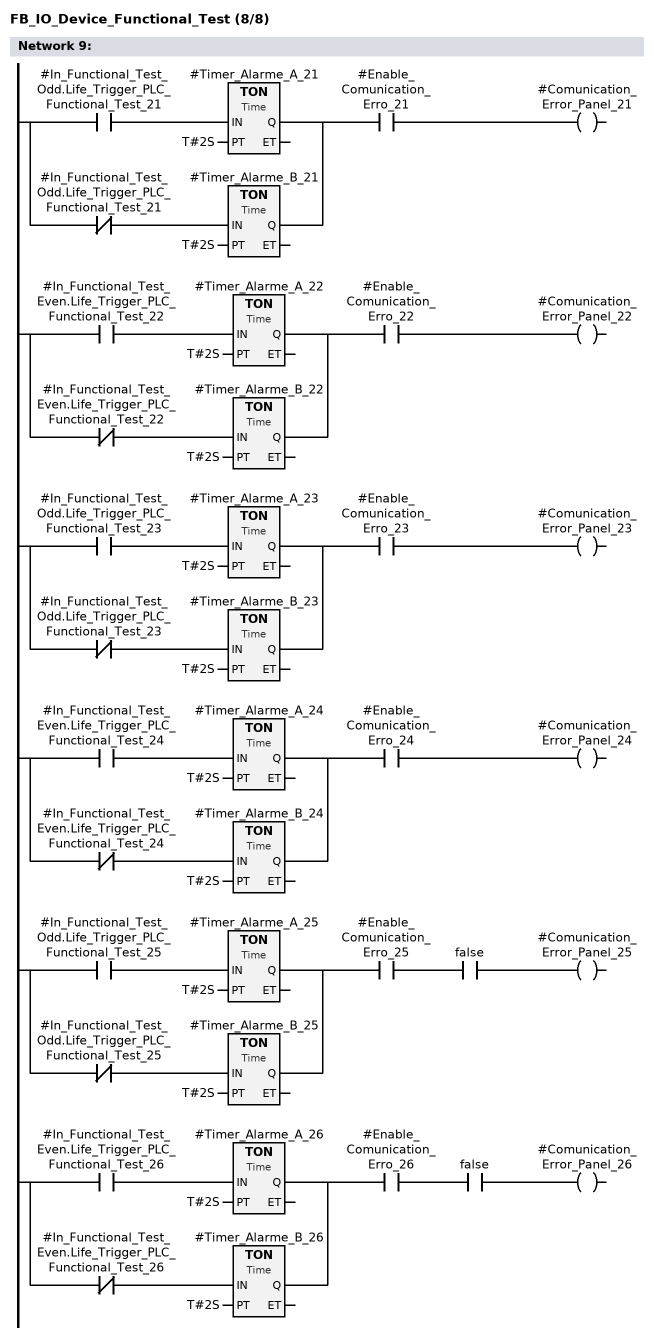
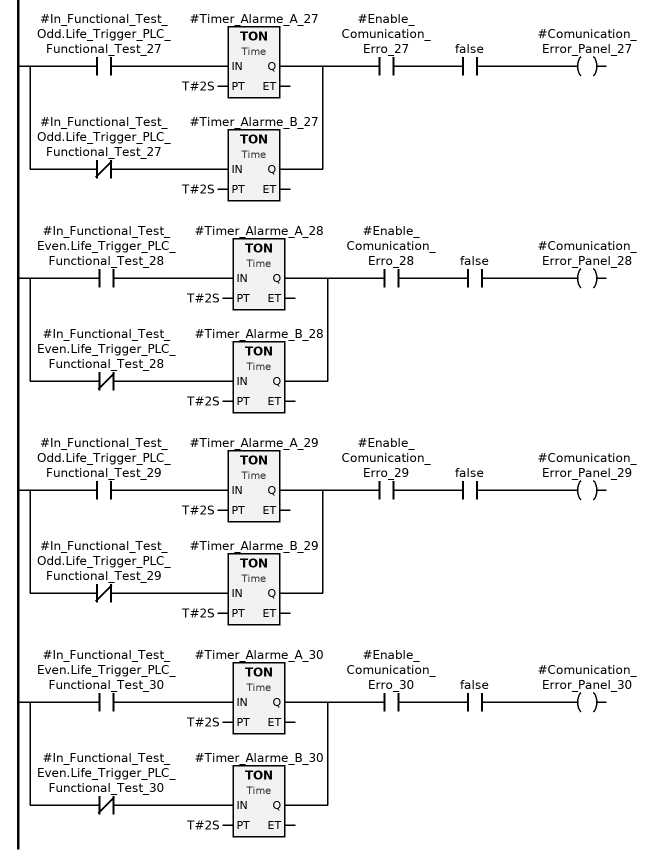
   RUNG wire#powerrail
      Contact( #In_Functional_Test_Odd.Life_Trigger_PLC_Functional_Test_21 )
      { S7_Templates := "time_type := Time" } #Timer_Alarme_A_21.TON(pt := T#2S, et =>)
      wire#w1
      Contact( #Enable_Comunication_Erro_21 )
      Coil( #Comunication_Error_Panel_21 )
   END_RUNG
   RUNG wire#powerrail
      I_Contact( #In_Functional_Test_Odd.Life_Trigger_PLC_Functional_Test_21 )
      { S7_Templates := "time_type := Time" } #Timer_Alarme_B_21.TON(pt := T#2S, et =>)
   END_RUNG wire#w1
   RUNG wire#powerrail
      Contact( #In_Functional_Test_Even.Life_Trigger_PLC_Functional_Test_22 )
      { S7_Templates := "time_type := Time" } #Timer_Alarme_A_22.TON(pt := T#2S, et =>)
      wire#w2
      Contact( #Enable_Comunication_Erro_22 )
      Coil( #Comunication_Error_Panel_22 )
   END_RUNG
   RUNG wire#powerrail
      I_Contact( #In_Functional_Test_Even.Life_Trigger_PLC_Functional_Test_22 )
      { S7_Templates := "time_type := Time" } #Timer_Alarme_B_22.TON(pt := T#2S, et =>)
   END_RUNG wire#w2
   RUNG wire#powerrail
      Contact( #In_Functional_Test_Odd.Life_Trigger_PLC_Functional_Test_23 )
      { S7_Templates := "time_type := Time" } #Timer_Alarme_A_23.TON(pt := T#2S, et =>)
      wire#w3
      Contact( #Enable_Comunication_Erro_23 )
      Coil( #Comunication_Error_Panel_23 )
   END_RUNG
   RUNG wire#powerrail
      I_Contact( #In_Functional_Test_Odd.Life_Trigger_PLC_Functional_Test_23 )
      { S7_Templates := "time_type := Time" } #Timer_Alarme_B_23.TON(pt := T#2S, et =>)
   END_RUNG wire#w3
   RUNG wire#powerrail
      Contact( #In_Functional_Test_Even.Life_Trigger_PLC_Functional_Test_24 )
      { S7_Templates := "time_type := Time" } #Timer_Alarme_A_24.TON(pt := T#2S, et =>)
      wire#w4
      Contact( #Enable_Comunication_Erro_24 )
      Coil( #Comunication_Error_Panel_24 )
   END_RUNG
   RUNG wire#powerrail
      I_Contact( #In_Functional_Test_Even.Life_Trigger_PLC_Functional_Test_24 )
      { S7_Templates := "time_type := Time" } #Timer_Alarme_B_24.TON(pt := T#2S, et =>)
   END_RUNG wire#w4
   RUNG wire#powerrail
      Contact( #In_Functional_Test_Odd.Life_Trigger_PLC_Functional_Test_25 )
      { S7_Templates := "time_type := Time" } #Timer_Alarme_A_25.TON(pt := T#2S, et =>)
      wire#w5
      Contact( #Enable_Comunication_Erro_25 )
      Contact( false )
      Coil( #Comunication_Error_Panel_25 )
   END_RUNG
   RUNG wire#powerrail
      I_Contact( #In_Functional_Test_Odd.Life_Trigger_PLC_Functional_Test_25 )
      { S7_Templates := "time_type := Time" } #Timer_Alarme_B_25.TON(pt := T#2S, et =>)
   END_RUNG wire#w5
   RUNG wire#powerrail
      Contact( #In_Functional_Test_Even.Life_Trigger_PLC_Functional_Test_26 )
      { S7_Templates := "time_type := Time" } #Timer_Alarme_A_26.TON(pt := T#2S, et =>)
      wire#w6
      Contact( #Enable_Comunication_Erro_26 )
      Contact( false )
      Coil( #Comunication_Error_Panel_26 )
   END_RUNG
   RUNG wire#powerrail
      I_Contact( #In_Functional_Test_Even.Life_Trigger_PLC_Functional_Test_26 )
      { S7_Templates := "time_type := Time" } #Timer_Alarme_B_26.TON(pt := T#2S, et =>)
   END_RUNG wire#w6
   RUNG wire#powerrail
      Contact( #In_Functional_Test_Odd.Life_Trigger_PLC_Functional_Test_27 )
      { S7_Templates := "time_type := Time" } #Timer_Alarme_A_27.TON(pt := T#2S, et =>)
      wire#w7
      Contact( #Enable_Comunication_Erro_27 )
      Contact( false )
      Coil( #Comunication_Error_Panel_27 )
   END_RUNG
   RUNG wire#powerrail
      I_Contact( #In_Functional_Test_Odd.Life_Trigger_PLC_Functional_Test_27 )
      { S7_Templates := "time_type := Time" } #Timer_Alarme_B_27.TON(pt := T#2S, et =>)
   END_RUNG wire#w7
   RUNG wire#powerrail
      Contact( #In_Functional_Test_Even.Life_Trigger_PLC_Functional_Test_28 )
      { S7_Templates := "time_type := Time" } #Timer_Alarme_A_28.TON(pt := T#2S, et =>)
      wire#w8
      Contact( #Enable_Comunication_Erro_28 )
      Contact( false )
      Coil( #Comunication_Error_Panel_28 )
   END_RUNG
   RUNG wire#powerrail
      I_Contact( #In_Functional_Test_Even.Life_Trigger_PLC_Functional_Test_28 )
      { S7_Templates := "time_type := Time" } #Timer_Alarme_B_28.TON(pt := T#2S, et =>)
   END_RUNG wire#w8
   RUNG wire#powerrail
      Contact( #In_Functional_Test_Odd.Life_Trigger_PLC_Functional_Test_29 )
      { S7_Templates := "time_type := Time" } #Timer_Alarme_A_29.TON(pt := T#2S, et =>)
      wire#w9
      Contact( #Enable_Comunication_Erro_29 )
      Contact( false )
      Coil( #Comunication_Error_Panel_29 )
   END_RUNG
   RUNG wire#powerrail
      I_Contact( #In_Functional_Test_Odd.Life_Trigger_PLC_Functional_Test_29 )
      { S7_Templates := "time_type := Time" } #Timer_Alarme_B_29.TON(pt := T#2S, et =>)
   END_RUNG wire#w9
   RUNG wire#powerrail
      Contact( #In_Functional_Test_Even.Life_Trigger_PLC_Functional_Test_30 )
      { S7_Templates := "time_type := Time" } #Timer_Alarme_A_30.TON(pt := T#2S, et =>)
      wire#w10
      Contact( #Enable_Comunication_Erro_30 )
      Contact( false )
      Coil( #Comunication_Error_Panel_30 )
   END_RUNG
   RUNG wire#powerrail
      I_Contact( #In_Functional_Test_Even.Life_Trigger_PLC_Functional_Test_30 )
      { S7_Templates := "time_type := Time" } #Timer_Alarme_B_30.TON(pt := T#2S, et =>)
   END_RUNG wire#w10
   // the same network as SCL:
   #Timer_Alarme_A_21(IN := #In_Functional_Test_Odd.Life_Trigger_PLC_Functional_Test_21, PT := T#2S);   // TON
   #Timer_Alarme_B_21(IN := NOT #In_Functional_Test_Odd.Life_Trigger_PLC_Functional_Test_21, PT := T#2S);   // TON
   #Comunication_Error_Panel_21 := (#Timer_Alarme_A_21.Q OR #Timer_Alarme_B_21.Q) AND #Enable_Comunication_Erro_21;
   #Timer_Alarme_A_22(IN := #In_Functional_Test_Even.Life_Trigger_PLC_Functional_Test_22, PT := T#2S);   // TON
   #Timer_Alarme_B_22(IN := NOT #In_Functional_Test_Even.Life_Trigger_PLC_Functional_Test_22, PT := T#2S);   // TON
   #Comunication_Error_Panel_22 := (#Timer_Alarme_A_22.Q OR #Timer_Alarme_B_22.Q) AND #Enable_Comunication_Erro_22;
   #Timer_Alarme_A_23(IN := #In_Functional_Test_Odd.Life_Trigger_PLC_Functional_Test_23, PT := T#2S);   // TON
   #Timer_Alarme_B_23(IN := NOT #In_Functional_Test_Odd.Life_Trigger_PLC_Functional_Test_23, PT := T#2S);   // TON
   #Comunication_Error_Panel_23 := (#Timer_Alarme_A_23.Q OR #Timer_Alarme_B_23.Q) AND #Enable_Comunication_Erro_23;
   #Timer_Alarme_A_24(IN := #In_Functional_Test_Even.Life_Trigger_PLC_Functional_Test_24, PT := T#2S);   // TON
   #Timer_Alarme_B_24(IN := NOT #In_Functional_Test_Even.Life_Trigger_PLC_Functional_Test_24, PT := T#2S);   // TON
   #Comunication_Error_Panel_24 := (#Timer_Alarme_A_24.Q OR #Timer_Alarme_B_24.Q) AND #Enable_Comunication_Erro_24;
   #Timer_Alarme_A_25(IN := #In_Functional_Test_Odd.Life_Trigger_PLC_Functional_Test_25, PT := T#2S);   // TON
   #Timer_Alarme_B_25(IN := NOT #In_Functional_Test_Odd.Life_Trigger_PLC_Functional_Test_25, PT := T#2S);   // TON
   #Comunication_Error_Panel_25 := (#Timer_Alarme_A_25.Q OR #Timer_Alarme_B_25.Q) AND #Enable_Comunication_Erro_25 AND false;
   #Timer_Alarme_A_26(IN := #In_Functional_Test_Even.Life_Trigger_PLC_Functional_Test_26, PT := T#2S);   // TON
   #Timer_Alarme_B_26(IN := NOT #In_Functional_Test_Even.Life_Trigger_PLC_Functional_Test_26, PT := T#2S);   // TON
   #Comunication_Error_Panel_26 := (#Timer_Alarme_A_26.Q OR #Timer_Alarme_B_26.Q) AND #Enable_Comunication_Erro_26 AND false;
   #Timer_Alarme_A_27(IN := #In_Functional_Test_Odd.Life_Trigger_PLC_Functional_Test_27, PT := T#2S);   // TON
   #Timer_Alarme_B_27(IN := NOT #In_Functional_Test_Odd.Life_Trigger_PLC_Functional_Test_27, PT := T#2S);   // TON
   #Comunication_Error_Panel_27 := (#Timer_Alarme_A_27.Q OR #Timer_Alarme_B_27.Q) AND #Enable_Comunication_Erro_27 AND false;
   #Timer_Alarme_A_28(IN := #In_Functional_Test_Even.Life_Trigger_PLC_Functional_Test_28, PT := T#2S);   // TON
   #Timer_Alarme_B_28(IN := NOT #In_Functional_Test_Even.Life_Trigger_PLC_Functional_Test_28, PT := T#2S);   // TON
   #Comunication_Error_Panel_28 := (#Timer_Alarme_A_28.Q OR #Timer_Alarme_B_28.Q) AND #Enable_Comunication_Erro_28 AND false;
   #Timer_Alarme_A_29(IN := #In_Functional_Test_Odd.Life_Trigger_PLC_Functional_Test_29, PT := T#2S);   // TON
   #Timer_Alarme_B_29(IN := NOT #In_Functional_Test_Odd.Life_Trigger_PLC_Functional_Test_29, PT := T#2S);   // TON
   #Comunication_Error_Panel_29 := (#Timer_Alarme_A_29.Q OR #Timer_Alarme_B_29.Q) AND #Enable_Comunication_Erro_29 AND false;
   #Timer_Alarme_A_30(IN := #In_Functional_Test_Even.Life_Trigger_PLC_Functional_Test_30, PT := T#2S);   // TON
   #Timer_Alarme_B_30(IN := NOT #In_Functional_Test_Even.Life_Trigger_PLC_Functional_Test_30, PT := T#2S);   // TON
   #Comunication_Error_Panel_30 := (#Timer_Alarme_A_30.Q OR #Timer_Alarme_B_30.Q) AND #Enable_Comunication_Erro_30 AND false;
END_REGION
END_FUNCTION_BLOCK

FUNCTION_BLOCK "FB_IO_Device_Production_And_Rework"   // FB5, LAD
{ S7_Optimized_Access := 'TRUE' }
// stored: MemoryReserve 100, SetENOAutomatically false
   VAR_INPUT
      Start : Bool;
      Manual_Turn_On_Motor_Caroussel : Bool;
      Manual_Turn_On_Motor_Conveyor_Belt : Bool;
      Water_Foutain_Fail_Functional_Test : Bool;
      Select_Motor_Speed : SInt;
      Carousel_Voltage_Selection : SInt;
      In_PLC_Production_And_Rework : "IO_Device_Conveyor_Belt_Input";
   END_VAR
   VAR_OUTPUT
      Comunication_Error : Bool;
      Emergency_Stop_Release : Bool;
      Trigger_Read_Serial_Number_Entrace_Functional_Test : Bool;
      Trigger_Read_Serial_Number_Exit_Functional_Test : Bool;
      Selected_Voltage_220V : Bool;
      Selected_Voltage_127V : Bool;
      Carousel_Frequency_Inverter_Fail : Bool;
      Conveyor_Belt_Functional_Test_Inverter_Fail : Bool;
      Out_PLC_Production_And_Rework : "IO_Device_Conveyor_Belt_Ouput";
   END_VAR
   VAR
      Timer_Alarme_A_1 { S7_SetPoint := 'True'} : TON_TIME;
      Timer_Alarme_B_1 { S7_SetPoint := 'True'} : TON_TIME;
   END_VAR
BEGIN

REGION Network 1
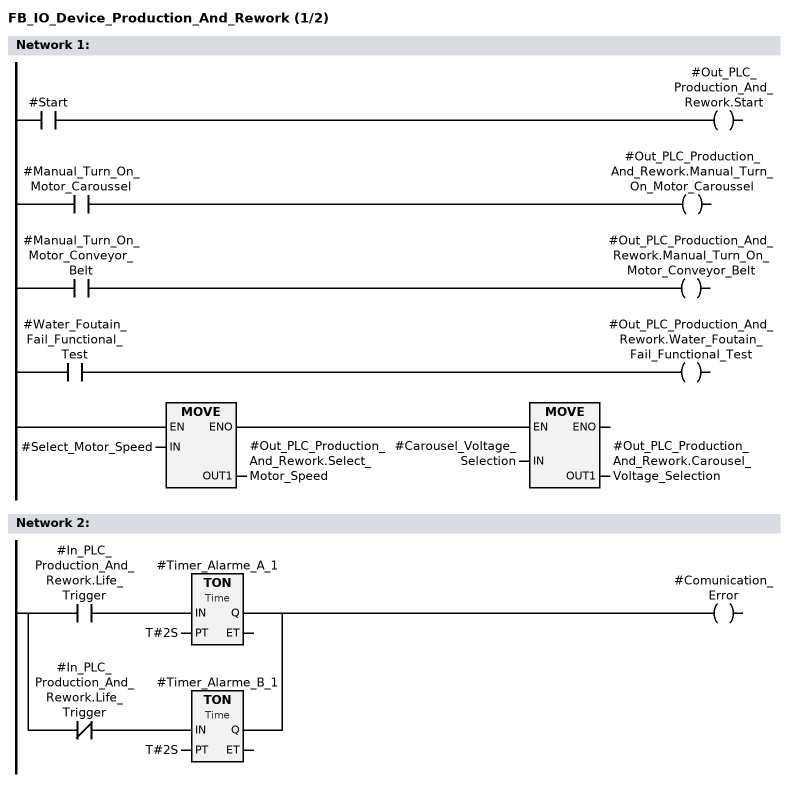
   RUNG wire#powerrail
      Contact( #Start )
      Coil( #Out_PLC_Production_And_Rework.Start )
   END_RUNG
   RUNG wire#powerrail
      Contact( #Manual_Turn_On_Motor_Caroussel )
      Coil( #Out_PLC_Production_And_Rework.Manual_Turn_On_Motor_Caroussel )
   END_RUNG
   RUNG wire#powerrail
      Contact( #Manual_Turn_On_Motor_Conveyor_Belt )
      Coil( #Out_PLC_Production_And_Rework.Manual_Turn_On_Motor_Conveyor_Belt )
   END_RUNG
   RUNG wire#powerrail
      Contact( #Water_Foutain_Fail_Functional_Test )
      Coil( #Out_PLC_Production_And_Rework.Water_Foutain_Fail_Functional_Test )
   END_RUNG
   RUNG wire#powerrail
      Move(in := #Select_Motor_Speed, out1 => #Out_PLC_Production_And_Rework.Select_Motor_Speed)
      Move(in := #Carousel_Voltage_Selection, out1 => #Out_PLC_Production_And_Rework.Carousel_Voltage_Selection)
   END_RUNG
   // the same network as SCL:
   #Out_PLC_Production_And_Rework.Start := #Start;
   #Out_PLC_Production_And_Rework.Manual_Turn_On_Motor_Caroussel := #Manual_Turn_On_Motor_Caroussel;
   #Out_PLC_Production_And_Rework.Manual_Turn_On_Motor_Conveyor_Belt := #Manual_Turn_On_Motor_Conveyor_Belt;
   #Out_PLC_Production_And_Rework.Water_Foutain_Fail_Functional_Test := #Water_Foutain_Fail_Functional_Test;
   #Out_PLC_Production_And_Rework.Select_Motor_Speed := #Select_Motor_Speed;
   #Out_PLC_Production_And_Rework.Carousel_Voltage_Selection := #Carousel_Voltage_Selection;
END_REGION

REGION Network 2
   RUNG wire#powerrail
      Contact( #In_PLC_Production_And_Rework.Life_Trigger )
      { S7_Templates := "time_type := Time" } #Timer_Alarme_A_1.TON(pt := T#2S, et =>)
      wire#w1
      Coil( #Comunication_Error )
   END_RUNG
   RUNG wire#powerrail
      I_Contact( #In_PLC_Production_And_Rework.Life_Trigger )
      { S7_Templates := "time_type := Time" } #Timer_Alarme_B_1.TON(pt := T#2S, et =>)
   END_RUNG wire#w1
   // the same network as SCL:
   #Timer_Alarme_A_1(IN := #In_PLC_Production_And_Rework.Life_Trigger, PT := T#2S);   // TON
   #Timer_Alarme_B_1(IN := NOT #In_PLC_Production_And_Rework.Life_Trigger, PT := T#2S);   // TON
   #Comunication_Error := #Timer_Alarme_A_1.Q OR #Timer_Alarme_B_1.Q;
END_REGION

REGION Network 3
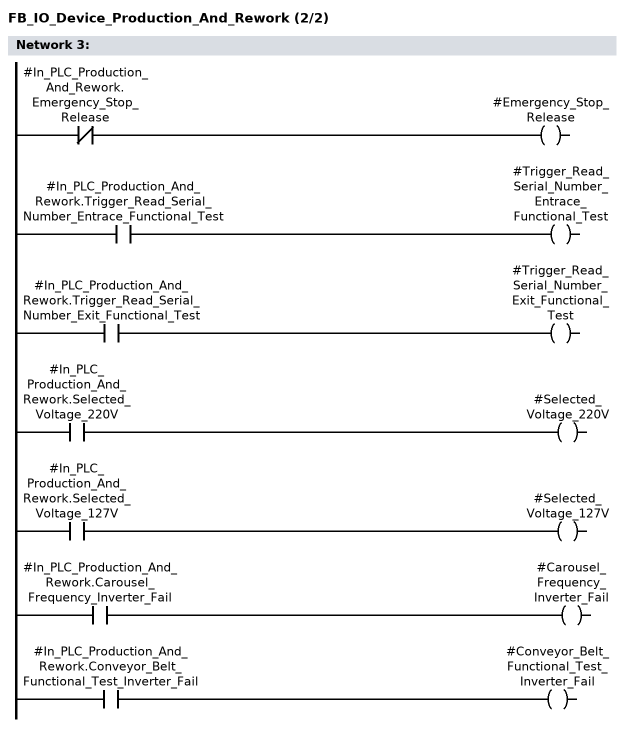
   RUNG wire#powerrail
      I_Contact( #In_PLC_Production_And_Rework.Emergency_Stop_Release )
      Coil( #Emergency_Stop_Release )
   END_RUNG
   RUNG wire#powerrail
      Contact( #In_PLC_Production_And_Rework.Trigger_Read_Serial_Number_Entrace_Functional_Test )
      Coil( #Trigger_Read_Serial_Number_Entrace_Functional_Test )
   END_RUNG
   RUNG wire#powerrail
      Contact( #In_PLC_Production_And_Rework.Trigger_Read_Serial_Number_Exit_Functional_Test )
      Coil( #Trigger_Read_Serial_Number_Exit_Functional_Test )
   END_RUNG
   RUNG wire#powerrail
      Contact( #In_PLC_Production_And_Rework.Selected_Voltage_220V )
      Coil( #Selected_Voltage_220V )
   END_RUNG
   RUNG wire#powerrail
      Contact( #In_PLC_Production_And_Rework.Selected_Voltage_127V )
      Coil( #Selected_Voltage_127V )
   END_RUNG
   RUNG wire#powerrail
      Contact( #In_PLC_Production_And_Rework.Carousel_Frequency_Inverter_Fail )
      Coil( #Carousel_Frequency_Inverter_Fail )
   END_RUNG
   RUNG wire#powerrail
      Contact( #In_PLC_Production_And_Rework.Conveyor_Belt_Functional_Test_Inverter_Fail )
      Coil( #Conveyor_Belt_Functional_Test_Inverter_Fail )
   END_RUNG
   // the same network as SCL:
   #Emergency_Stop_Release := NOT #In_PLC_Production_And_Rework.Emergency_Stop_Release;
   #Trigger_Read_Serial_Number_Entrace_Functional_Test := #In_PLC_Production_And_Rework.Trigger_Read_Serial_Number_Entrace_Functional_Test;
   #Trigger_Read_Serial_Number_Exit_Functional_Test := #In_PLC_Production_And_Rework.Trigger_Read_Serial_Number_Exit_Functional_Test;
   #Selected_Voltage_220V := #In_PLC_Production_And_Rework.Selected_Voltage_220V;
   #Selected_Voltage_127V := #In_PLC_Production_And_Rework.Selected_Voltage_127V;
   #Carousel_Frequency_Inverter_Fail := #In_PLC_Production_And_Rework.Carousel_Frequency_Inverter_Fail;
   #Conveyor_Belt_Functional_Test_Inverter_Fail := #In_PLC_Production_And_Rework.Conveyor_Belt_Functional_Test_Inverter_Fail;
END_REGION
END_FUNCTION_BLOCK

FUNCTION_BLOCK "FB_Read_Data_SR-X100W"   // FB6, LAD
{ S7_Optimized_Access := 'TRUE' }
// stored: AutoNumber false, MemoryReserve 100, SetENOAutomatically false
   VAR_INPUT
      Trigger_Sensor : Bool;
      Read_Complete : Bool;
      Read_Failure : Bool;
      Clear_Data : Bool;
      Read_Data_In : "SR-X100W_Read_Data";
   END_VAR
   VAR_OUTPUT
      Read_Request : Bool;
      Read_Complete_Clear : Bool;
      Read_Complete_OUT : Bool;
      Read_Failure_OUT : Bool;
      Read_Data_Out : String[136];
      Serial_Number { ExternalAccessible := 'False'; ExternalVisible := 'False'; ExternalWritable := 'False'} : String[17];
   END_VAR
   VAR
      Aux_Triggger_1 : Bool;
      Aux_Triggger_2 : Bool;
      Aux_Triggger_3 : Bool;
      Aux_Triggger_4 : Bool;
      DB_What_Was_Read_Instance { S7_SetPoint := 'True'} : "FB_What_Was_Read";
      Timer_Delay_Reset { S7_SetPoint := 'True'} : TON_TIME;
   END_VAR
   VAR_TEMP   // added for the SCL form of the ladder/FBD networks
      _w1 : Bool;
      _w2 : Bool;
   END_VAR
BEGIN

REGION Network 1
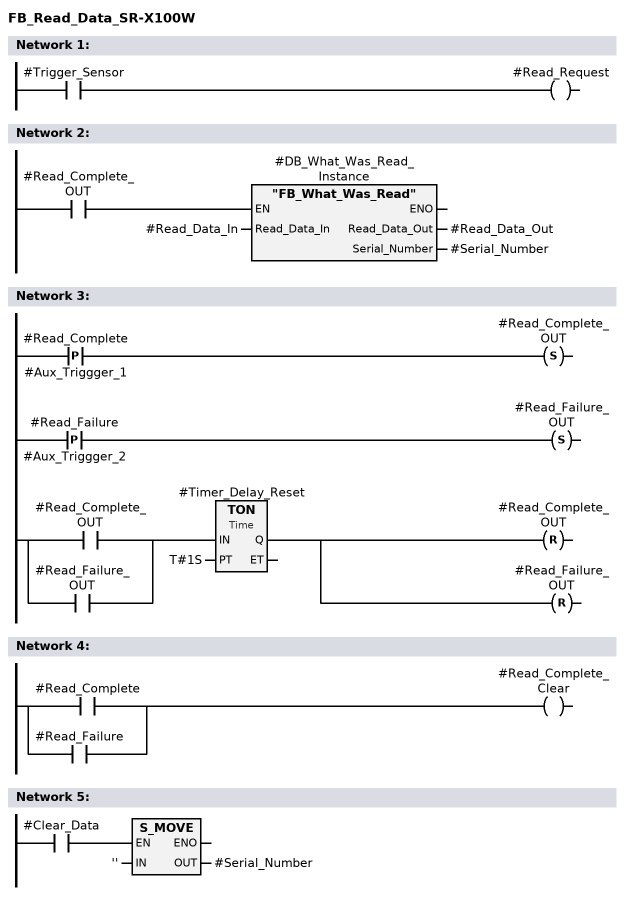
   RUNG wire#powerrail
      Contact( #Trigger_Sensor )
      Coil( #Read_Request )
   END_RUNG
   // the same network as SCL:
   #Read_Request := #Trigger_Sensor;
END_REGION

REGION Network 2
   RUNG wire#powerrail
      Contact( #Read_Complete_OUT )
      #DB_What_Was_Read_Instance(Read_Data_In := #Read_Data_In, Read_Data_Out => #Read_Data_Out, Serial_Number => #Serial_Number)
   END_RUNG
   // the same network as SCL:
   IF #Read_Complete_OUT THEN
       #DB_What_Was_Read_Instance(Read_Data_In := #Read_Data_In,   // "FB_What_Was_Read"
                               Read_Data_Out => #Read_Data_Out,
                               Serial_Number => #Serial_Number);
   END_IF;
END_REGION

REGION Network 3
   RUNG wire#powerrail
      P_Contact(operand := #Read_Complete, bit := #Aux_Triggger_1)
      S_Coil( #Read_Complete_OUT )
   END_RUNG
   RUNG wire#powerrail
      P_Contact(operand := #Read_Failure, bit := #Aux_Triggger_2)
      S_Coil( #Read_Failure_OUT )
   END_RUNG
   RUNG wire#powerrail
      Contact( #Read_Complete_OUT )
      wire#w1
      { S7_Templates := "time_type := Time" } #Timer_Delay_Reset.TON(pt := T#1S, et =>)
      wire#w2
      R_Coil( #Read_Complete_OUT )
   END_RUNG
   RUNG wire#powerrail
      Contact( #Read_Failure_OUT )
   END_RUNG wire#w1
   RUNG wire#w2
      R_Coil( #Read_Failure_OUT )
   END_RUNG
   // the same network as SCL:
   #_w1 := #Read_Complete AND NOT #Aux_Triggger_1;   // rising edge of #Read_Complete
   #Aux_Triggger_1 := #Read_Complete;
   IF #_w1 THEN #Read_Complete_OUT := TRUE; END_IF;
   #_w2 := #Read_Failure AND NOT #Aux_Triggger_2;   // rising edge of #Read_Failure
   #Aux_Triggger_2 := #Read_Failure;
   IF #_w2 THEN #Read_Failure_OUT := TRUE; END_IF;
   #Timer_Delay_Reset(IN := #Read_Complete_OUT OR #Read_Failure_OUT, PT := T#1S);   // TON
   IF #Timer_Delay_Reset.Q THEN
       #Read_Complete_OUT := FALSE;
       #Read_Failure_OUT := FALSE;
   END_IF;
END_REGION

REGION Network 4
   RUNG wire#powerrail
      Contact( #Read_Complete )
      wire#w1
      Coil( #Read_Complete_Clear )
   END_RUNG
   RUNG wire#powerrail
      Contact( #Read_Failure )
   END_RUNG wire#w1
   // the same network as SCL:
   #Read_Complete_Clear := #Read_Complete OR #Read_Failure;
END_REGION

REGION Network 5
   RUNG wire#powerrail
      Contact( #Clear_Data )
      S_Move(in := '', out => #Serial_Number)
   END_RUNG
   // the same network as SCL:
   IF #Clear_Data THEN #Serial_Number := ''; END_IF;
END_REGION
END_FUNCTION_BLOCK

FUNCTION_BLOCK "FB_What_Was_Read"   // FB7, LAD
{ S7_Optimized_Access := 'TRUE' }
// stored: AutoNumber false, MemoryReserve 100, SetENOAutomatically false
   VAR_INPUT
      Read_Data_In : "SR-X100W_Read_Data";
   END_VAR
   VAR_OUTPUT
      Read_Data_Out : String[136];
      Serial_Number : String[17];
   END_VAR
BEGIN

REGION Network 1
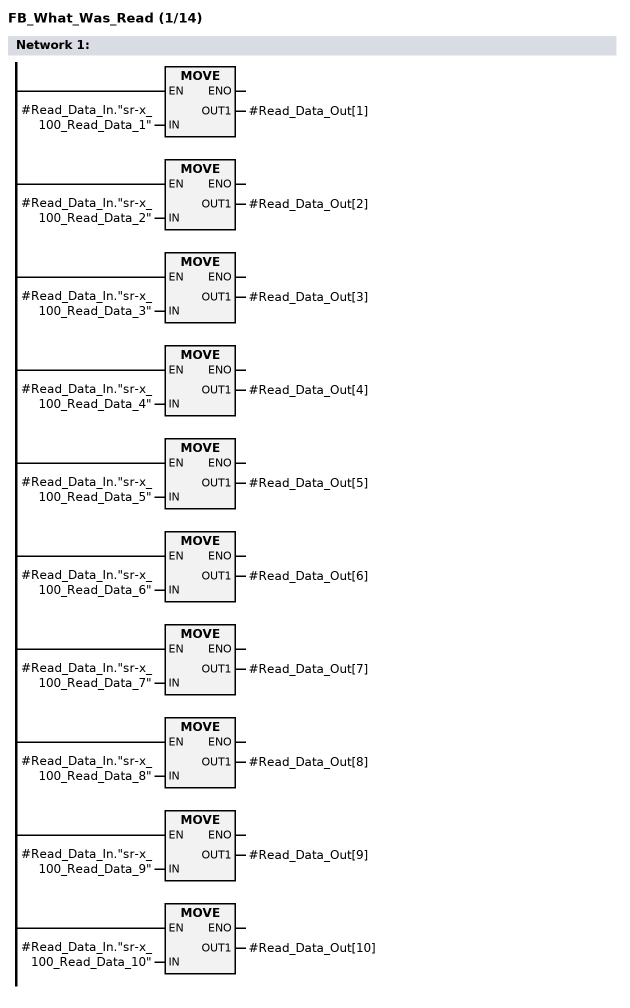
   RUNG wire#powerrail
      Move(in := #Read_Data_In."sr-x_100_Read_Data_1", out1 => #Read_Data_Out[1])
   END_RUNG
   RUNG wire#powerrail
      Move(in := #Read_Data_In."sr-x_100_Read_Data_2", out1 => #Read_Data_Out[2])
   END_RUNG
   RUNG wire#powerrail
      Move(in := #Read_Data_In."sr-x_100_Read_Data_3", out1 => #Read_Data_Out[3])
   END_RUNG
   RUNG wire#powerrail
      Move(in := #Read_Data_In."sr-x_100_Read_Data_4", out1 => #Read_Data_Out[4])
   END_RUNG
   RUNG wire#powerrail
      Move(in := #Read_Data_In."sr-x_100_Read_Data_5", out1 => #Read_Data_Out[5])
   END_RUNG
   RUNG wire#powerrail
      Move(in := #Read_Data_In."sr-x_100_Read_Data_6", out1 => #Read_Data_Out[6])
   END_RUNG
   RUNG wire#powerrail
      Move(in := #Read_Data_In."sr-x_100_Read_Data_7", out1 => #Read_Data_Out[7])
   END_RUNG
   RUNG wire#powerrail
      Move(in := #Read_Data_In."sr-x_100_Read_Data_8", out1 => #Read_Data_Out[8])
   END_RUNG
   RUNG wire#powerrail
      Move(in := #Read_Data_In."sr-x_100_Read_Data_9", out1 => #Read_Data_Out[9])
   END_RUNG
   RUNG wire#powerrail
      Move(in := #Read_Data_In."sr-x_100_Read_Data_10", out1 => #Read_Data_Out[10])
   END_RUNG
   // the same network as SCL:
   #Read_Data_Out[1] := #Read_Data_In."sr-x_100_Read_Data_1";
   #Read_Data_Out[2] := #Read_Data_In."sr-x_100_Read_Data_2";
   #Read_Data_Out[3] := #Read_Data_In."sr-x_100_Read_Data_3";
   #Read_Data_Out[4] := #Read_Data_In."sr-x_100_Read_Data_4";
   #Read_Data_Out[5] := #Read_Data_In."sr-x_100_Read_Data_5";
   #Read_Data_Out[6] := #Read_Data_In."sr-x_100_Read_Data_6";
   #Read_Data_Out[7] := #Read_Data_In."sr-x_100_Read_Data_7";
   #Read_Data_Out[8] := #Read_Data_In."sr-x_100_Read_Data_8";
   #Read_Data_Out[9] := #Read_Data_In."sr-x_100_Read_Data_9";
   #Read_Data_Out[10] := #Read_Data_In."sr-x_100_Read_Data_10";
END_REGION

REGION Network 2
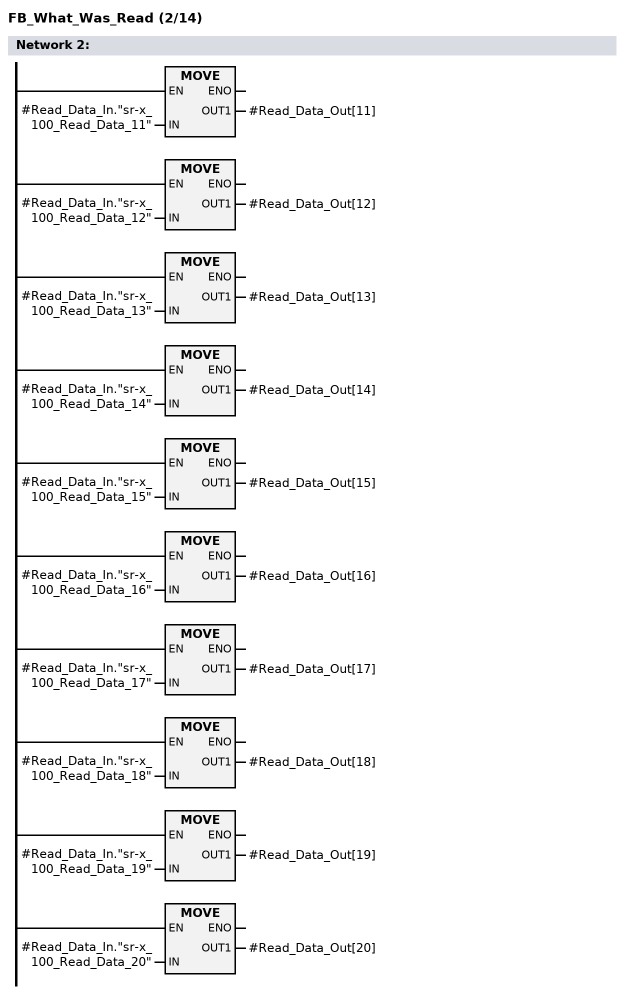
   RUNG wire#powerrail
      Move(in := #Read_Data_In."sr-x_100_Read_Data_11", out1 => #Read_Data_Out[11])
   END_RUNG
   RUNG wire#powerrail
      Move(in := #Read_Data_In."sr-x_100_Read_Data_12", out1 => #Read_Data_Out[12])
   END_RUNG
   RUNG wire#powerrail
      Move(in := #Read_Data_In."sr-x_100_Read_Data_13", out1 => #Read_Data_Out[13])
   END_RUNG
   RUNG wire#powerrail
      Move(in := #Read_Data_In."sr-x_100_Read_Data_14", out1 => #Read_Data_Out[14])
   END_RUNG
   RUNG wire#powerrail
      Move(in := #Read_Data_In."sr-x_100_Read_Data_15", out1 => #Read_Data_Out[15])
   END_RUNG
   RUNG wire#powerrail
      Move(in := #Read_Data_In."sr-x_100_Read_Data_16", out1 => #Read_Data_Out[16])
   END_RUNG
   RUNG wire#powerrail
      Move(in := #Read_Data_In."sr-x_100_Read_Data_17", out1 => #Read_Data_Out[17])
   END_RUNG
   RUNG wire#powerrail
      Move(in := #Read_Data_In."sr-x_100_Read_Data_18", out1 => #Read_Data_Out[18])
   END_RUNG
   RUNG wire#powerrail
      Move(in := #Read_Data_In."sr-x_100_Read_Data_19", out1 => #Read_Data_Out[19])
   END_RUNG
   RUNG wire#powerrail
      Move(in := #Read_Data_In."sr-x_100_Read_Data_20", out1 => #Read_Data_Out[20])
   END_RUNG
   // the same network as SCL:
   #Read_Data_Out[11] := #Read_Data_In."sr-x_100_Read_Data_11";
   #Read_Data_Out[12] := #Read_Data_In."sr-x_100_Read_Data_12";
   #Read_Data_Out[13] := #Read_Data_In."sr-x_100_Read_Data_13";
   #Read_Data_Out[14] := #Read_Data_In."sr-x_100_Read_Data_14";
   #Read_Data_Out[15] := #Read_Data_In."sr-x_100_Read_Data_15";
   #Read_Data_Out[16] := #Read_Data_In."sr-x_100_Read_Data_16";
   #Read_Data_Out[17] := #Read_Data_In."sr-x_100_Read_Data_17";
   #Read_Data_Out[18] := #Read_Data_In."sr-x_100_Read_Data_18";
   #Read_Data_Out[19] := #Read_Data_In."sr-x_100_Read_Data_19";
   #Read_Data_Out[20] := #Read_Data_In."sr-x_100_Read_Data_20";
END_REGION

REGION Network 3
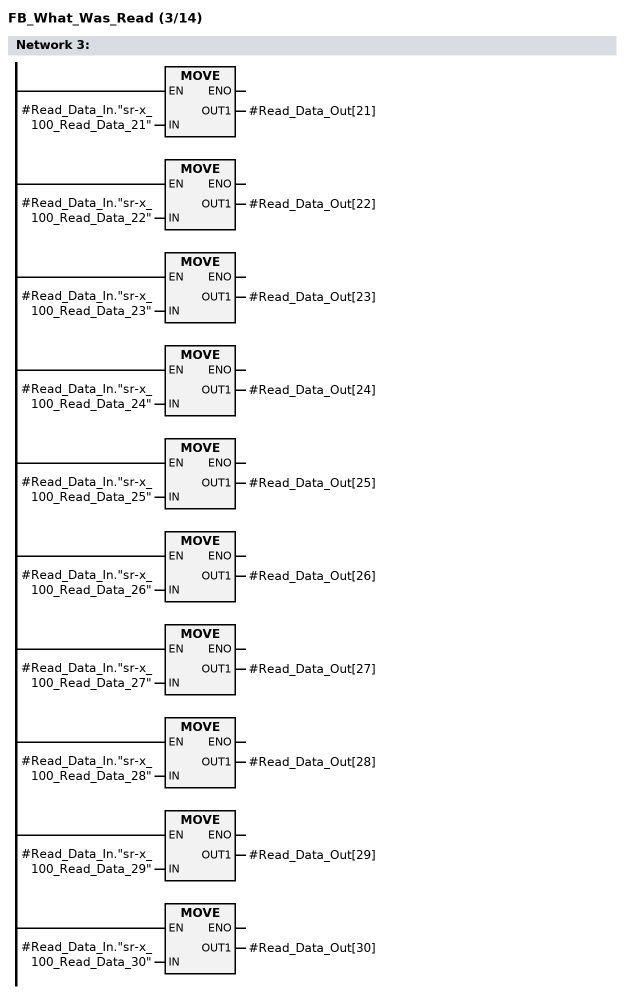
   RUNG wire#powerrail
      Move(in := #Read_Data_In."sr-x_100_Read_Data_21", out1 => #Read_Data_Out[21])
   END_RUNG
   RUNG wire#powerrail
      Move(in := #Read_Data_In."sr-x_100_Read_Data_22", out1 => #Read_Data_Out[22])
   END_RUNG
   RUNG wire#powerrail
      Move(in := #Read_Data_In."sr-x_100_Read_Data_23", out1 => #Read_Data_Out[23])
   END_RUNG
   RUNG wire#powerrail
      Move(in := #Read_Data_In."sr-x_100_Read_Data_24", out1 => #Read_Data_Out[24])
   END_RUNG
   RUNG wire#powerrail
      Move(in := #Read_Data_In."sr-x_100_Read_Data_25", out1 => #Read_Data_Out[25])
   END_RUNG
   RUNG wire#powerrail
      Move(in := #Read_Data_In."sr-x_100_Read_Data_26", out1 => #Read_Data_Out[26])
   END_RUNG
   RUNG wire#powerrail
      Move(in := #Read_Data_In."sr-x_100_Read_Data_27", out1 => #Read_Data_Out[27])
   END_RUNG
   RUNG wire#powerrail
      Move(in := #Read_Data_In."sr-x_100_Read_Data_28", out1 => #Read_Data_Out[28])
   END_RUNG
   RUNG wire#powerrail
      Move(in := #Read_Data_In."sr-x_100_Read_Data_29", out1 => #Read_Data_Out[29])
   END_RUNG
   RUNG wire#powerrail
      Move(in := #Read_Data_In."sr-x_100_Read_Data_30", out1 => #Read_Data_Out[30])
   END_RUNG
   // the same network as SCL:
   #Read_Data_Out[21] := #Read_Data_In."sr-x_100_Read_Data_21";
   #Read_Data_Out[22] := #Read_Data_In."sr-x_100_Read_Data_22";
   #Read_Data_Out[23] := #Read_Data_In."sr-x_100_Read_Data_23";
   #Read_Data_Out[24] := #Read_Data_In."sr-x_100_Read_Data_24";
   #Read_Data_Out[25] := #Read_Data_In."sr-x_100_Read_Data_25";
   #Read_Data_Out[26] := #Read_Data_In."sr-x_100_Read_Data_26";
   #Read_Data_Out[27] := #Read_Data_In."sr-x_100_Read_Data_27";
   #Read_Data_Out[28] := #Read_Data_In."sr-x_100_Read_Data_28";
   #Read_Data_Out[29] := #Read_Data_In."sr-x_100_Read_Data_29";
   #Read_Data_Out[30] := #Read_Data_In."sr-x_100_Read_Data_30";
END_REGION

REGION Network 4
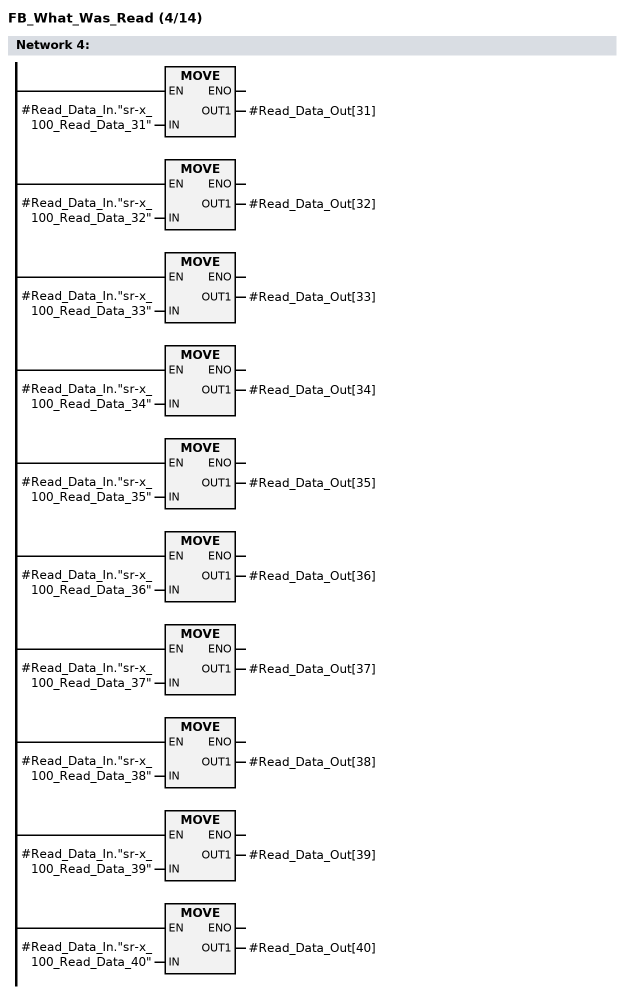
   RUNG wire#powerrail
      Move(in := #Read_Data_In."sr-x_100_Read_Data_31", out1 => #Read_Data_Out[31])
   END_RUNG
   RUNG wire#powerrail
      Move(in := #Read_Data_In."sr-x_100_Read_Data_32", out1 => #Read_Data_Out[32])
   END_RUNG
   RUNG wire#powerrail
      Move(in := #Read_Data_In."sr-x_100_Read_Data_33", out1 => #Read_Data_Out[33])
   END_RUNG
   RUNG wire#powerrail
      Move(in := #Read_Data_In."sr-x_100_Read_Data_34", out1 => #Read_Data_Out[34])
   END_RUNG
   RUNG wire#powerrail
      Move(in := #Read_Data_In."sr-x_100_Read_Data_35", out1 => #Read_Data_Out[35])
   END_RUNG
   RUNG wire#powerrail
      Move(in := #Read_Data_In."sr-x_100_Read_Data_36", out1 => #Read_Data_Out[36])
   END_RUNG
   RUNG wire#powerrail
      Move(in := #Read_Data_In."sr-x_100_Read_Data_37", out1 => #Read_Data_Out[37])
   END_RUNG
   RUNG wire#powerrail
      Move(in := #Read_Data_In."sr-x_100_Read_Data_38", out1 => #Read_Data_Out[38])
   END_RUNG
   RUNG wire#powerrail
      Move(in := #Read_Data_In."sr-x_100_Read_Data_39", out1 => #Read_Data_Out[39])
   END_RUNG
   RUNG wire#powerrail
      Move(in := #Read_Data_In."sr-x_100_Read_Data_40", out1 => #Read_Data_Out[40])
   END_RUNG
   // the same network as SCL:
   #Read_Data_Out[31] := #Read_Data_In."sr-x_100_Read_Data_31";
   #Read_Data_Out[32] := #Read_Data_In."sr-x_100_Read_Data_32";
   #Read_Data_Out[33] := #Read_Data_In."sr-x_100_Read_Data_33";
   #Read_Data_Out[34] := #Read_Data_In."sr-x_100_Read_Data_34";
   #Read_Data_Out[35] := #Read_Data_In."sr-x_100_Read_Data_35";
   #Read_Data_Out[36] := #Read_Data_In."sr-x_100_Read_Data_36";
   #Read_Data_Out[37] := #Read_Data_In."sr-x_100_Read_Data_37";
   #Read_Data_Out[38] := #Read_Data_In."sr-x_100_Read_Data_38";
   #Read_Data_Out[39] := #Read_Data_In."sr-x_100_Read_Data_39";
   #Read_Data_Out[40] := #Read_Data_In."sr-x_100_Read_Data_40";
END_REGION

REGION Network 5
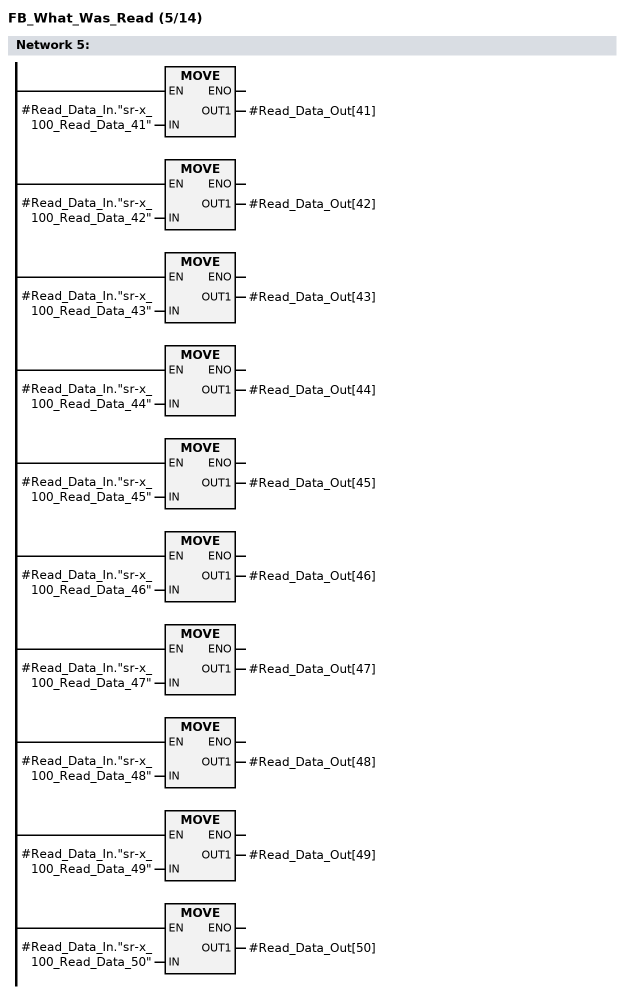
   RUNG wire#powerrail
      Move(in := #Read_Data_In."sr-x_100_Read_Data_41", out1 => #Read_Data_Out[41])
   END_RUNG
   RUNG wire#powerrail
      Move(in := #Read_Data_In."sr-x_100_Read_Data_42", out1 => #Read_Data_Out[42])
   END_RUNG
   RUNG wire#powerrail
      Move(in := #Read_Data_In."sr-x_100_Read_Data_43", out1 => #Read_Data_Out[43])
   END_RUNG
   RUNG wire#powerrail
      Move(in := #Read_Data_In."sr-x_100_Read_Data_44", out1 => #Read_Data_Out[44])
   END_RUNG
   RUNG wire#powerrail
      Move(in := #Read_Data_In."sr-x_100_Read_Data_45", out1 => #Read_Data_Out[45])
   END_RUNG
   RUNG wire#powerrail
      Move(in := #Read_Data_In."sr-x_100_Read_Data_46", out1 => #Read_Data_Out[46])
   END_RUNG
   RUNG wire#powerrail
      Move(in := #Read_Data_In."sr-x_100_Read_Data_47", out1 => #Read_Data_Out[47])
   END_RUNG
   RUNG wire#powerrail
      Move(in := #Read_Data_In."sr-x_100_Read_Data_48", out1 => #Read_Data_Out[48])
   END_RUNG
   RUNG wire#powerrail
      Move(in := #Read_Data_In."sr-x_100_Read_Data_49", out1 => #Read_Data_Out[49])
   END_RUNG
   RUNG wire#powerrail
      Move(in := #Read_Data_In."sr-x_100_Read_Data_50", out1 => #Read_Data_Out[50])
   END_RUNG
   // the same network as SCL:
   #Read_Data_Out[41] := #Read_Data_In."sr-x_100_Read_Data_41";
   #Read_Data_Out[42] := #Read_Data_In."sr-x_100_Read_Data_42";
   #Read_Data_Out[43] := #Read_Data_In."sr-x_100_Read_Data_43";
   #Read_Data_Out[44] := #Read_Data_In."sr-x_100_Read_Data_44";
   #Read_Data_Out[45] := #Read_Data_In."sr-x_100_Read_Data_45";
   #Read_Data_Out[46] := #Read_Data_In."sr-x_100_Read_Data_46";
   #Read_Data_Out[47] := #Read_Data_In."sr-x_100_Read_Data_47";
   #Read_Data_Out[48] := #Read_Data_In."sr-x_100_Read_Data_48";
   #Read_Data_Out[49] := #Read_Data_In."sr-x_100_Read_Data_49";
   #Read_Data_Out[50] := #Read_Data_In."sr-x_100_Read_Data_50";
END_REGION

REGION Network 6
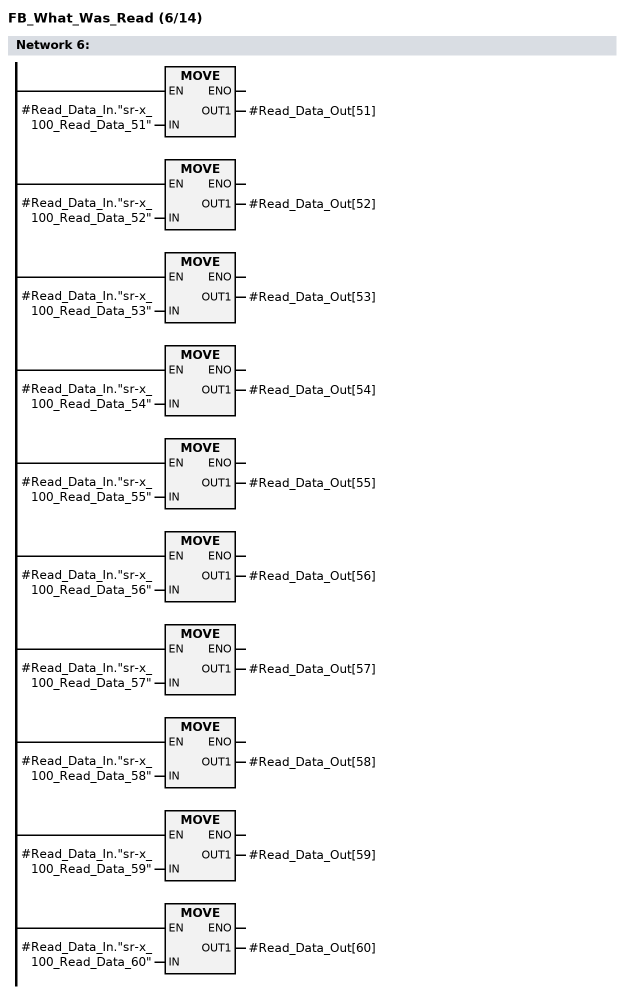
   RUNG wire#powerrail
      Move(in := #Read_Data_In."sr-x_100_Read_Data_51", out1 => #Read_Data_Out[51])
   END_RUNG
   RUNG wire#powerrail
      Move(in := #Read_Data_In."sr-x_100_Read_Data_52", out1 => #Read_Data_Out[52])
   END_RUNG
   RUNG wire#powerrail
      Move(in := #Read_Data_In."sr-x_100_Read_Data_53", out1 => #Read_Data_Out[53])
   END_RUNG
   RUNG wire#powerrail
      Move(in := #Read_Data_In."sr-x_100_Read_Data_54", out1 => #Read_Data_Out[54])
   END_RUNG
   RUNG wire#powerrail
      Move(in := #Read_Data_In."sr-x_100_Read_Data_55", out1 => #Read_Data_Out[55])
   END_RUNG
   RUNG wire#powerrail
      Move(in := #Read_Data_In."sr-x_100_Read_Data_56", out1 => #Read_Data_Out[56])
   END_RUNG
   RUNG wire#powerrail
      Move(in := #Read_Data_In."sr-x_100_Read_Data_57", out1 => #Read_Data_Out[57])
   END_RUNG
   RUNG wire#powerrail
      Move(in := #Read_Data_In."sr-x_100_Read_Data_58", out1 => #Read_Data_Out[58])
   END_RUNG
   RUNG wire#powerrail
      Move(in := #Read_Data_In."sr-x_100_Read_Data_59", out1 => #Read_Data_Out[59])
   END_RUNG
   RUNG wire#powerrail
      Move(in := #Read_Data_In."sr-x_100_Read_Data_60", out1 => #Read_Data_Out[60])
   END_RUNG
   // the same network as SCL:
   #Read_Data_Out[51] := #Read_Data_In."sr-x_100_Read_Data_51";
   #Read_Data_Out[52] := #Read_Data_In."sr-x_100_Read_Data_52";
   #Read_Data_Out[53] := #Read_Data_In."sr-x_100_Read_Data_53";
   #Read_Data_Out[54] := #Read_Data_In."sr-x_100_Read_Data_54";
   #Read_Data_Out[55] := #Read_Data_In."sr-x_100_Read_Data_55";
   #Read_Data_Out[56] := #Read_Data_In."sr-x_100_Read_Data_56";
   #Read_Data_Out[57] := #Read_Data_In."sr-x_100_Read_Data_57";
   #Read_Data_Out[58] := #Read_Data_In."sr-x_100_Read_Data_58";
   #Read_Data_Out[59] := #Read_Data_In."sr-x_100_Read_Data_59";
   #Read_Data_Out[60] := #Read_Data_In."sr-x_100_Read_Data_60";
END_REGION

REGION Network 7
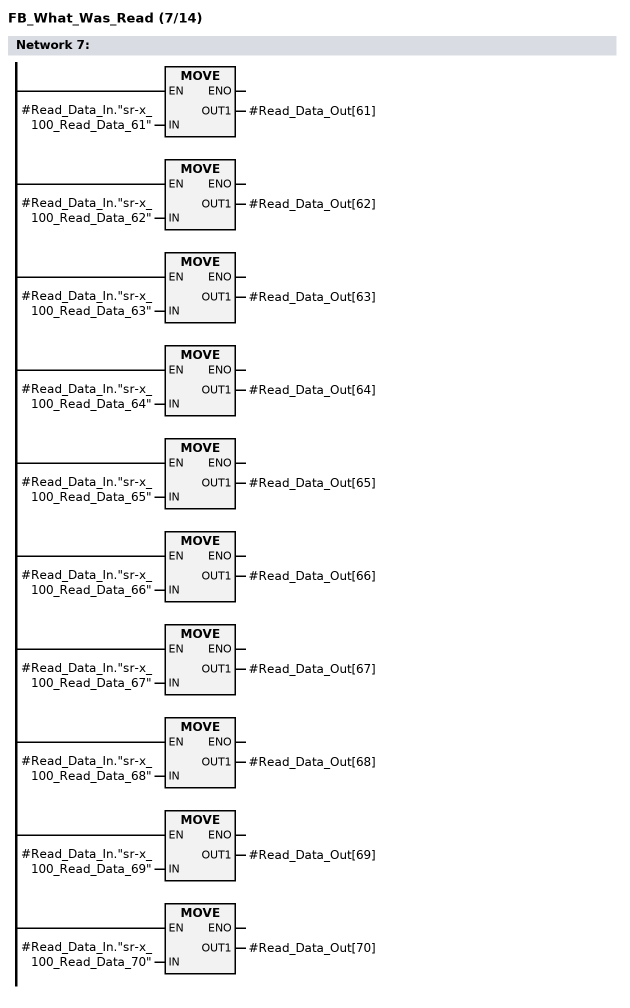
   RUNG wire#powerrail
      Move(in := #Read_Data_In."sr-x_100_Read_Data_61", out1 => #Read_Data_Out[61])
   END_RUNG
   RUNG wire#powerrail
      Move(in := #Read_Data_In."sr-x_100_Read_Data_62", out1 => #Read_Data_Out[62])
   END_RUNG
   RUNG wire#powerrail
      Move(in := #Read_Data_In."sr-x_100_Read_Data_63", out1 => #Read_Data_Out[63])
   END_RUNG
   RUNG wire#powerrail
      Move(in := #Read_Data_In."sr-x_100_Read_Data_64", out1 => #Read_Data_Out[64])
   END_RUNG
   RUNG wire#powerrail
      Move(in := #Read_Data_In."sr-x_100_Read_Data_65", out1 => #Read_Data_Out[65])
   END_RUNG
   RUNG wire#powerrail
      Move(in := #Read_Data_In."sr-x_100_Read_Data_66", out1 => #Read_Data_Out[66])
   END_RUNG
   RUNG wire#powerrail
      Move(in := #Read_Data_In."sr-x_100_Read_Data_67", out1 => #Read_Data_Out[67])
   END_RUNG
   RUNG wire#powerrail
      Move(in := #Read_Data_In."sr-x_100_Read_Data_68", out1 => #Read_Data_Out[68])
   END_RUNG
   RUNG wire#powerrail
      Move(in := #Read_Data_In."sr-x_100_Read_Data_69", out1 => #Read_Data_Out[69])
   END_RUNG
   RUNG wire#powerrail
      Move(in := #Read_Data_In."sr-x_100_Read_Data_70", out1 => #Read_Data_Out[70])
   END_RUNG
   // the same network as SCL:
   #Read_Data_Out[61] := #Read_Data_In."sr-x_100_Read_Data_61";
   #Read_Data_Out[62] := #Read_Data_In."sr-x_100_Read_Data_62";
   #Read_Data_Out[63] := #Read_Data_In."sr-x_100_Read_Data_63";
   #Read_Data_Out[64] := #Read_Data_In."sr-x_100_Read_Data_64";
   #Read_Data_Out[65] := #Read_Data_In."sr-x_100_Read_Data_65";
   #Read_Data_Out[66] := #Read_Data_In."sr-x_100_Read_Data_66";
   #Read_Data_Out[67] := #Read_Data_In."sr-x_100_Read_Data_67";
   #Read_Data_Out[68] := #Read_Data_In."sr-x_100_Read_Data_68";
   #Read_Data_Out[69] := #Read_Data_In."sr-x_100_Read_Data_69";
   #Read_Data_Out[70] := #Read_Data_In."sr-x_100_Read_Data_70";
END_REGION

REGION Network 8
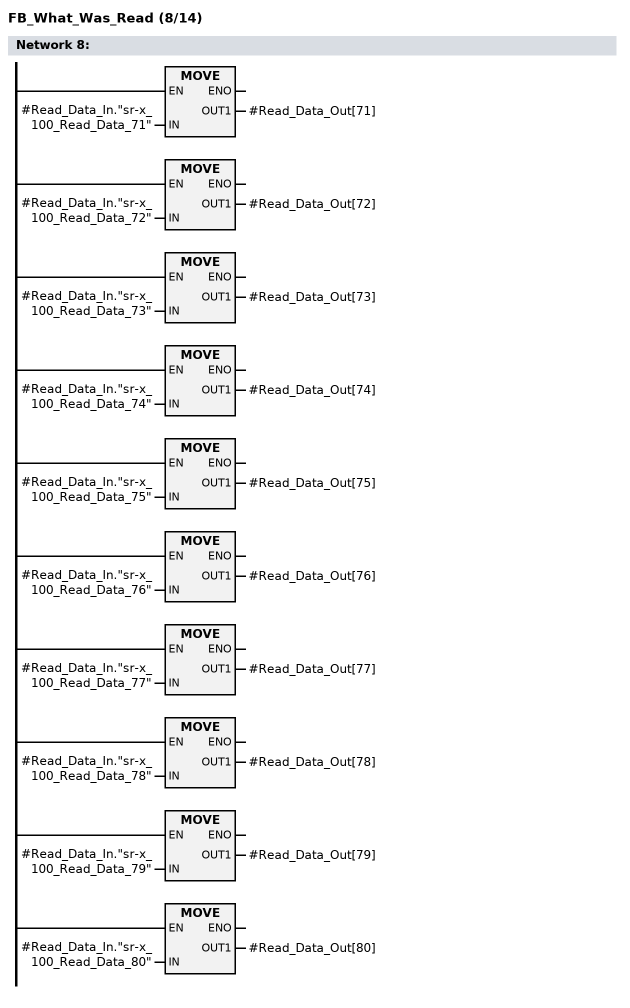
   RUNG wire#powerrail
      Move(in := #Read_Data_In."sr-x_100_Read_Data_71", out1 => #Read_Data_Out[71])
   END_RUNG
   RUNG wire#powerrail
      Move(in := #Read_Data_In."sr-x_100_Read_Data_72", out1 => #Read_Data_Out[72])
   END_RUNG
   RUNG wire#powerrail
      Move(in := #Read_Data_In."sr-x_100_Read_Data_73", out1 => #Read_Data_Out[73])
   END_RUNG
   RUNG wire#powerrail
      Move(in := #Read_Data_In."sr-x_100_Read_Data_74", out1 => #Read_Data_Out[74])
   END_RUNG
   RUNG wire#powerrail
      Move(in := #Read_Data_In."sr-x_100_Read_Data_75", out1 => #Read_Data_Out[75])
   END_RUNG
   RUNG wire#powerrail
      Move(in := #Read_Data_In."sr-x_100_Read_Data_76", out1 => #Read_Data_Out[76])
   END_RUNG
   RUNG wire#powerrail
      Move(in := #Read_Data_In."sr-x_100_Read_Data_77", out1 => #Read_Data_Out[77])
   END_RUNG
   RUNG wire#powerrail
      Move(in := #Read_Data_In."sr-x_100_Read_Data_78", out1 => #Read_Data_Out[78])
   END_RUNG
   RUNG wire#powerrail
      Move(in := #Read_Data_In."sr-x_100_Read_Data_79", out1 => #Read_Data_Out[79])
   END_RUNG
   RUNG wire#powerrail
      Move(in := #Read_Data_In."sr-x_100_Read_Data_80", out1 => #Read_Data_Out[80])
   END_RUNG
   // the same network as SCL:
   #Read_Data_Out[71] := #Read_Data_In."sr-x_100_Read_Data_71";
   #Read_Data_Out[72] := #Read_Data_In."sr-x_100_Read_Data_72";
   #Read_Data_Out[73] := #Read_Data_In."sr-x_100_Read_Data_73";
   #Read_Data_Out[74] := #Read_Data_In."sr-x_100_Read_Data_74";
   #Read_Data_Out[75] := #Read_Data_In."sr-x_100_Read_Data_75";
   #Read_Data_Out[76] := #Read_Data_In."sr-x_100_Read_Data_76";
   #Read_Data_Out[77] := #Read_Data_In."sr-x_100_Read_Data_77";
   #Read_Data_Out[78] := #Read_Data_In."sr-x_100_Read_Data_78";
   #Read_Data_Out[79] := #Read_Data_In."sr-x_100_Read_Data_79";
   #Read_Data_Out[80] := #Read_Data_In."sr-x_100_Read_Data_80";
END_REGION

REGION Network 9
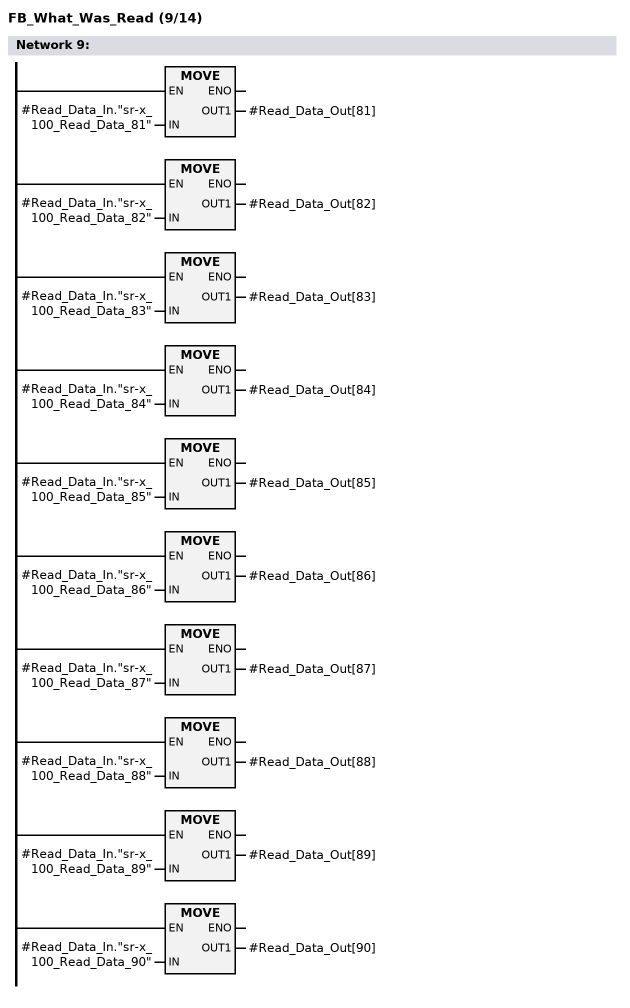
   RUNG wire#powerrail
      Move(in := #Read_Data_In."sr-x_100_Read_Data_81", out1 => #Read_Data_Out[81])
   END_RUNG
   RUNG wire#powerrail
      Move(in := #Read_Data_In."sr-x_100_Read_Data_82", out1 => #Read_Data_Out[82])
   END_RUNG
   RUNG wire#powerrail
      Move(in := #Read_Data_In."sr-x_100_Read_Data_83", out1 => #Read_Data_Out[83])
   END_RUNG
   RUNG wire#powerrail
      Move(in := #Read_Data_In."sr-x_100_Read_Data_84", out1 => #Read_Data_Out[84])
   END_RUNG
   RUNG wire#powerrail
      Move(in := #Read_Data_In."sr-x_100_Read_Data_85", out1 => #Read_Data_Out[85])
   END_RUNG
   RUNG wire#powerrail
      Move(in := #Read_Data_In."sr-x_100_Read_Data_86", out1 => #Read_Data_Out[86])
   END_RUNG
   RUNG wire#powerrail
      Move(in := #Read_Data_In."sr-x_100_Read_Data_87", out1 => #Read_Data_Out[87])
   END_RUNG
   RUNG wire#powerrail
      Move(in := #Read_Data_In."sr-x_100_Read_Data_88", out1 => #Read_Data_Out[88])
   END_RUNG
   RUNG wire#powerrail
      Move(in := #Read_Data_In."sr-x_100_Read_Data_89", out1 => #Read_Data_Out[89])
   END_RUNG
   RUNG wire#powerrail
      Move(in := #Read_Data_In."sr-x_100_Read_Data_90", out1 => #Read_Data_Out[90])
   END_RUNG
   // the same network as SCL:
   #Read_Data_Out[81] := #Read_Data_In."sr-x_100_Read_Data_81";
   #Read_Data_Out[82] := #Read_Data_In."sr-x_100_Read_Data_82";
   #Read_Data_Out[83] := #Read_Data_In."sr-x_100_Read_Data_83";
   #Read_Data_Out[84] := #Read_Data_In."sr-x_100_Read_Data_84";
   #Read_Data_Out[85] := #Read_Data_In."sr-x_100_Read_Data_85";
   #Read_Data_Out[86] := #Read_Data_In."sr-x_100_Read_Data_86";
   #Read_Data_Out[87] := #Read_Data_In."sr-x_100_Read_Data_87";
   #Read_Data_Out[88] := #Read_Data_In."sr-x_100_Read_Data_88";
   #Read_Data_Out[89] := #Read_Data_In."sr-x_100_Read_Data_89";
   #Read_Data_Out[90] := #Read_Data_In."sr-x_100_Read_Data_90";
END_REGION

REGION Network 10
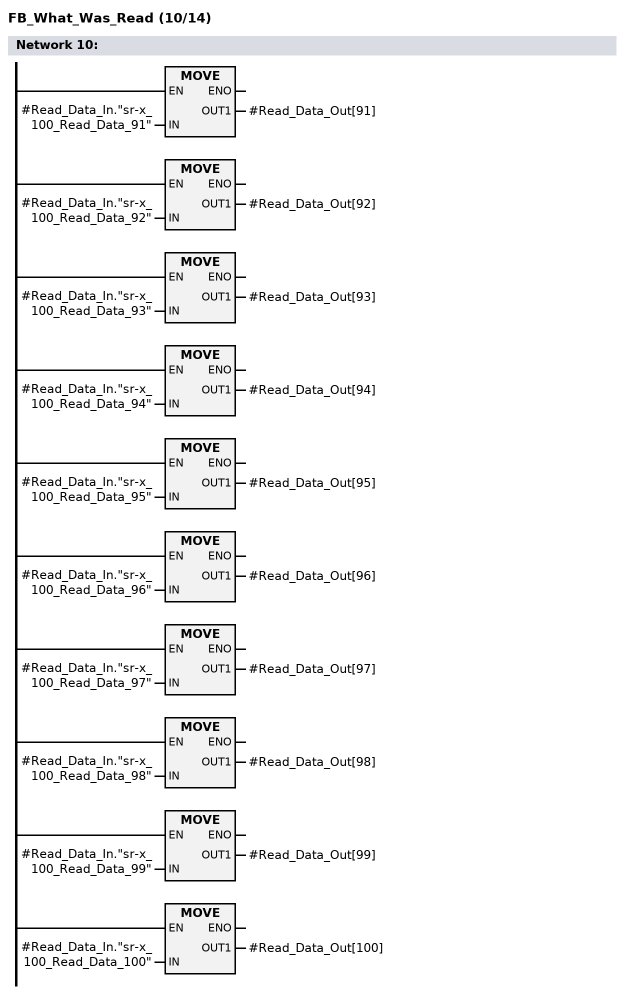
   RUNG wire#powerrail
      Move(in := #Read_Data_In."sr-x_100_Read_Data_91", out1 => #Read_Data_Out[91])
   END_RUNG
   RUNG wire#powerrail
      Move(in := #Read_Data_In."sr-x_100_Read_Data_92", out1 => #Read_Data_Out[92])
   END_RUNG
   RUNG wire#powerrail
      Move(in := #Read_Data_In."sr-x_100_Read_Data_93", out1 => #Read_Data_Out[93])
   END_RUNG
   RUNG wire#powerrail
      Move(in := #Read_Data_In."sr-x_100_Read_Data_94", out1 => #Read_Data_Out[94])
   END_RUNG
   RUNG wire#powerrail
      Move(in := #Read_Data_In."sr-x_100_Read_Data_95", out1 => #Read_Data_Out[95])
   END_RUNG
   RUNG wire#powerrail
      Move(in := #Read_Data_In."sr-x_100_Read_Data_96", out1 => #Read_Data_Out[96])
   END_RUNG
   RUNG wire#powerrail
      Move(in := #Read_Data_In."sr-x_100_Read_Data_97", out1 => #Read_Data_Out[97])
   END_RUNG
   RUNG wire#powerrail
      Move(in := #Read_Data_In."sr-x_100_Read_Data_98", out1 => #Read_Data_Out[98])
   END_RUNG
   RUNG wire#powerrail
      Move(in := #Read_Data_In."sr-x_100_Read_Data_99", out1 => #Read_Data_Out[99])
   END_RUNG
   RUNG wire#powerrail
      Move(in := #Read_Data_In."sr-x_100_Read_Data_100", out1 => #Read_Data_Out[100])
   END_RUNG
   // the same network as SCL:
   #Read_Data_Out[91] := #Read_Data_In."sr-x_100_Read_Data_91";
   #Read_Data_Out[92] := #Read_Data_In."sr-x_100_Read_Data_92";
   #Read_Data_Out[93] := #Read_Data_In."sr-x_100_Read_Data_93";
   #Read_Data_Out[94] := #Read_Data_In."sr-x_100_Read_Data_94";
   #Read_Data_Out[95] := #Read_Data_In."sr-x_100_Read_Data_95";
   #Read_Data_Out[96] := #Read_Data_In."sr-x_100_Read_Data_96";
   #Read_Data_Out[97] := #Read_Data_In."sr-x_100_Read_Data_97";
   #Read_Data_Out[98] := #Read_Data_In."sr-x_100_Read_Data_98";
   #Read_Data_Out[99] := #Read_Data_In."sr-x_100_Read_Data_99";
   #Read_Data_Out[100] := #Read_Data_In."sr-x_100_Read_Data_100";
END_REGION

REGION Network 11
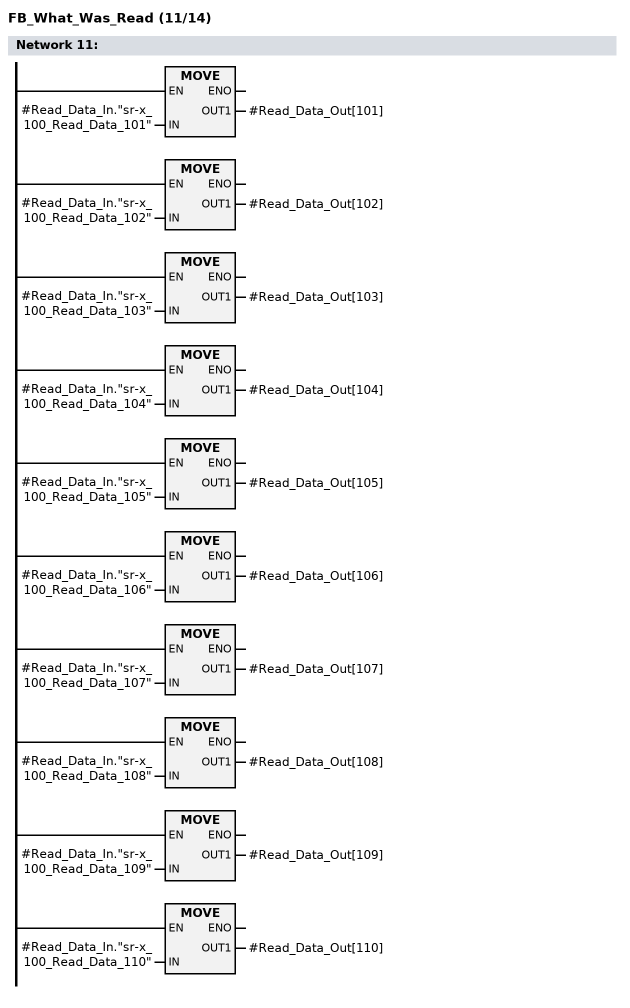
   RUNG wire#powerrail
      Move(in := #Read_Data_In."sr-x_100_Read_Data_101", out1 => #Read_Data_Out[101])
   END_RUNG
   RUNG wire#powerrail
      Move(in := #Read_Data_In."sr-x_100_Read_Data_102", out1 => #Read_Data_Out[102])
   END_RUNG
   RUNG wire#powerrail
      Move(in := #Read_Data_In."sr-x_100_Read_Data_103", out1 => #Read_Data_Out[103])
   END_RUNG
   RUNG wire#powerrail
      Move(in := #Read_Data_In."sr-x_100_Read_Data_104", out1 => #Read_Data_Out[104])
   END_RUNG
   RUNG wire#powerrail
      Move(in := #Read_Data_In."sr-x_100_Read_Data_105", out1 => #Read_Data_Out[105])
   END_RUNG
   RUNG wire#powerrail
      Move(in := #Read_Data_In."sr-x_100_Read_Data_106", out1 => #Read_Data_Out[106])
   END_RUNG
   RUNG wire#powerrail
      Move(in := #Read_Data_In."sr-x_100_Read_Data_107", out1 => #Read_Data_Out[107])
   END_RUNG
   RUNG wire#powerrail
      Move(in := #Read_Data_In."sr-x_100_Read_Data_108", out1 => #Read_Data_Out[108])
   END_RUNG
   RUNG wire#powerrail
      Move(in := #Read_Data_In."sr-x_100_Read_Data_109", out1 => #Read_Data_Out[109])
   END_RUNG
   RUNG wire#powerrail
      Move(in := #Read_Data_In."sr-x_100_Read_Data_110", out1 => #Read_Data_Out[110])
   END_RUNG
   // the same network as SCL:
   #Read_Data_Out[101] := #Read_Data_In."sr-x_100_Read_Data_101";
   #Read_Data_Out[102] := #Read_Data_In."sr-x_100_Read_Data_102";
   #Read_Data_Out[103] := #Read_Data_In."sr-x_100_Read_Data_103";
   #Read_Data_Out[104] := #Read_Data_In."sr-x_100_Read_Data_104";
   #Read_Data_Out[105] := #Read_Data_In."sr-x_100_Read_Data_105";
   #Read_Data_Out[106] := #Read_Data_In."sr-x_100_Read_Data_106";
   #Read_Data_Out[107] := #Read_Data_In."sr-x_100_Read_Data_107";
   #Read_Data_Out[108] := #Read_Data_In."sr-x_100_Read_Data_108";
   #Read_Data_Out[109] := #Read_Data_In."sr-x_100_Read_Data_109";
   #Read_Data_Out[110] := #Read_Data_In."sr-x_100_Read_Data_110";
END_REGION

REGION Network 12
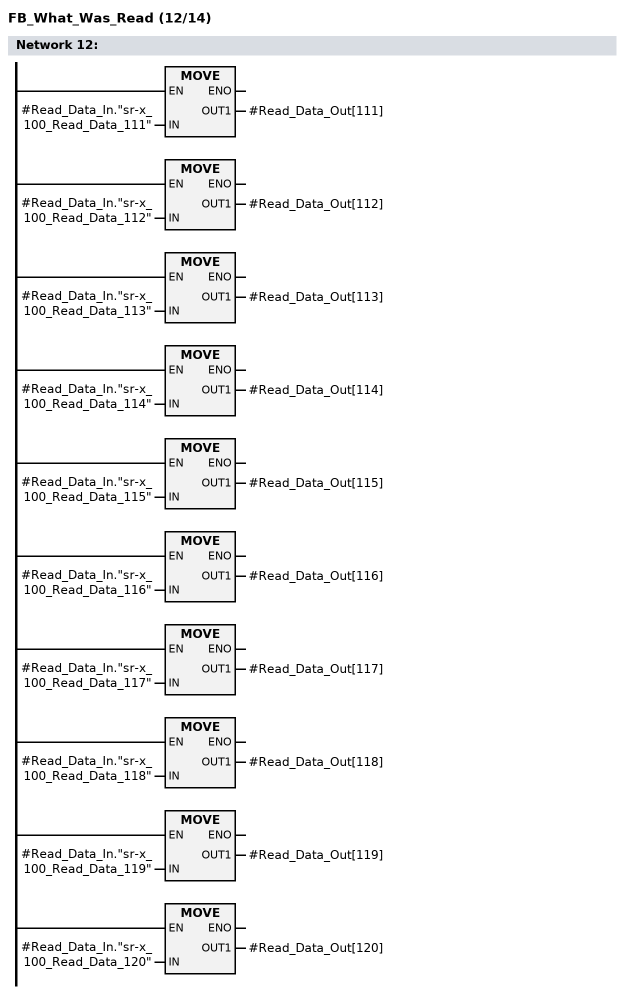
   RUNG wire#powerrail
      Move(in := #Read_Data_In."sr-x_100_Read_Data_111", out1 => #Read_Data_Out[111])
   END_RUNG
   RUNG wire#powerrail
      Move(in := #Read_Data_In."sr-x_100_Read_Data_112", out1 => #Read_Data_Out[112])
   END_RUNG
   RUNG wire#powerrail
      Move(in := #Read_Data_In."sr-x_100_Read_Data_113", out1 => #Read_Data_Out[113])
   END_RUNG
   RUNG wire#powerrail
      Move(in := #Read_Data_In."sr-x_100_Read_Data_114", out1 => #Read_Data_Out[114])
   END_RUNG
   RUNG wire#powerrail
      Move(in := #Read_Data_In."sr-x_100_Read_Data_115", out1 => #Read_Data_Out[115])
   END_RUNG
   RUNG wire#powerrail
      Move(in := #Read_Data_In."sr-x_100_Read_Data_116", out1 => #Read_Data_Out[116])
   END_RUNG
   RUNG wire#powerrail
      Move(in := #Read_Data_In."sr-x_100_Read_Data_117", out1 => #Read_Data_Out[117])
   END_RUNG
   RUNG wire#powerrail
      Move(in := #Read_Data_In."sr-x_100_Read_Data_118", out1 => #Read_Data_Out[118])
   END_RUNG
   RUNG wire#powerrail
      Move(in := #Read_Data_In."sr-x_100_Read_Data_119", out1 => #Read_Data_Out[119])
   END_RUNG
   RUNG wire#powerrail
      Move(in := #Read_Data_In."sr-x_100_Read_Data_120", out1 => #Read_Data_Out[120])
   END_RUNG
   // the same network as SCL:
   #Read_Data_Out[111] := #Read_Data_In."sr-x_100_Read_Data_111";
   #Read_Data_Out[112] := #Read_Data_In."sr-x_100_Read_Data_112";
   #Read_Data_Out[113] := #Read_Data_In."sr-x_100_Read_Data_113";
   #Read_Data_Out[114] := #Read_Data_In."sr-x_100_Read_Data_114";
   #Read_Data_Out[115] := #Read_Data_In."sr-x_100_Read_Data_115";
   #Read_Data_Out[116] := #Read_Data_In."sr-x_100_Read_Data_116";
   #Read_Data_Out[117] := #Read_Data_In."sr-x_100_Read_Data_117";
   #Read_Data_Out[118] := #Read_Data_In."sr-x_100_Read_Data_118";
   #Read_Data_Out[119] := #Read_Data_In."sr-x_100_Read_Data_119";
   #Read_Data_Out[120] := #Read_Data_In."sr-x_100_Read_Data_120";
END_REGION

REGION Network 13
